LIN {X 0,Y 573.253,Z 273.707,A -85,B 0,C 180,E1 -2292.186,E2 -2292.186} C_VEL
LIN {X 0,Y 573.222,Z 273.707,A -85,B 0,C 180,E1 -2294.675,E2 -2294.675} C_VEL
LIN {X 0,Y 573.232,Z 273.706,A -85,B 0,C 180,E1 -2297.599,E2 -2297.599} C_VEL
LIN {X 0,Y 573.243,Z 273.707,A -85,B 0,C 180,E1 -2300.393,E2 -2300.393} C_VEL
LIN {X 0,Y 573.246,Z 273.706,A -85,B 0,C 180,E1 -2303.077,E2 -2303.077} C_VEL
LIN {X 0,Y 573.254,Z 273.702,A -85,B 0,C 180,E1 -2305.671,E2 -2305.671} C_VEL
LIN {X 0,Y 573.242,Z 273.706,A -85,B 0,C 180,E1 -2308.185,E2 -2308.185} C_VEL
LIN {X 0,Y 573.254,Z 273.705,A -85,B 0,C 180,E1 -2310.634,E2 -2310.634} C_VEL
LIN {X 0,Y 573.228,Z 273.706,A -85,B 0,C 180,E1 -2313.507,E2 -2313.507} C_VEL
LIN {X 0,Y 573.225,Z 273.705,A -85,B 0,C 180,E1 -2316.134,E2 -2316.134} C_VEL
LIN {X 0,Y 573.238,Z 273.704,A -85,B 0,C 180,E1 -2319.173,E2 -2319.173} C_VEL
LIN {X 0,Y 573.23,Z 273.707,A -85,B 0,C 180,E1 -2321.412,E2 -2321.412} C_VEL
LIN {X 0,Y 573.243,Z 273.704,A -85,B 0,C 180,E1 -2323.622,E2 -2323.622} C_VEL
LIN {X 0,Y 573.216,Z 273.708,A -85,B 0,C 180,E1 -2326.529,E2 -2326.529} C_VEL
LIN {X 0,Y 573.275,Z 273.699,A -85,B 0,C 180,E1 -2328.734,E2 -2328.734} C_VEL
LIN {X 0,Y 573.276,Z 273.698,A -85,B 0,C 180,E1 -2331.54,E2 -2331.54} C_VEL
LIN {X 0,Y 573.283,Z 273.698,A -85,B 0,C 180,E1 -2334.372,E2 -2334.372} C_VEL
LIN {X 0,Y 573.31,Z 273.694,A -85,B 0,C 180,E1 -2337.892,E2 -2337.892} C_VEL
LIN {X 0,Y 573.31,Z 273.695,A -85,B 0,C 180,E1 -2340.702,E2 -2340.702} C_VEL
LIN {X 0,Y 573.298,Z 273.699,A -85,B 0,C 180,E1 -2342.811,E2 -2342.811} C_VEL
LIN {X 0,Y 573.283,Z 273.699,A -85,B 0,C 180,E1 -2345.628,E2 -2345.628} C_VEL
LIN {X 0,Y 573.276,Z 273.698,A -85,B 0,C 180,E1 -2348.46,E2 -2348.46} C_VEL
LIN {X 0,Y 573.262,Z 273.7,A -85,B 0,C 180,E1 -2351.312,E2 -2351.312} C_VEL
LIN {X 0,Y 573.247,Z 273.703,A -85,B 0,C 180,E1 -2354.194,E2 -2354.194} C_VEL
LIN {X 0,Y 573.251,Z 273.704,A -85,B 0,C 180,E1 -2357.112,E2 -2357.112} C_VEL
LIN {X 0,Y 573.238,Z 273.707,A -85,B 0,C 180,E1 -2360.077,E2 -2360.077} C_VEL
LIN {X 0,Y 573.226,Z 273.705,A -85,B 0,C 180,E1 -2362.338,E2 -2362.338} C_VEL
LIN {X 0,Y 573.242,Z 273.704,A -85,B 0,C 180,E1 -2364.372,E2 -2364.372} C_VEL
LIN {X 0,Y 572.615,Z 273.786,A -85,B 0,C 180,E1 -2364.958,E2 -2364.958} C_VEL
LIN {X 0,Y 569.777,Z 274.144,A -85,B 0,C 180,E1 -2365.91,E2 -2365.91} C_VEL
LIN {X 0,Y 567.344,Z 274.445,A -85,B 0,C 180,E1 -2366.675,E2 -2366.675} C_VEL
LIN {X 0,Y 566.282,Z 274.573,A -85,B 0,C 180,E1 -2367.266,E2 -2367.266} C_VEL
LIN {X 0,Y 566.188,Z 274.583,A -85,B 0,C 180,E1 -2367.466,E2 -2367.466} C_VEL
LIN {X 0,Y 566.194,Z 274.58,A -85,B 0,C 180,E1 -2369.769,E2 -2369.769} C_VEL
LIN {X 0,Y 566.201,Z 274.582,A -85,B 0,C 180,E1 -2372.431,E2 -2372.431} C_VEL
LIN {X 0,Y 566.163,Z 274.588,A -85,B 0,C 180,E1 -2374.989,E2 -2374.989} C_VEL
LIN {X 0,Y 566.191,Z 274.581,A -85,B 0,C 180,E1 -2377.461,E2 -2377.461} C_VEL
LIN {X 0,Y 566.213,Z 274.58,A -85,B 0,C 180,E1 -2380.199,E2 -2380.199} C_VEL
LIN {X 0,Y 566.195,Z 274.584,A -85,B 0,C 180,E1 -2383.055,E2 -2383.055} C_VEL
LIN {X 0,Y 566.198,Z 274.586,A -85,B 0,C 180,E1 -2386.049,E2 -2386.049} C_VEL
LIN {X 0,Y 566.161,Z 274.589,A -85,B 0,C 180,E1 -2388.143,E2 -2388.143} C_VEL
LIN {X 0,Y 566.274,Z 277.89,A -85,B 0,C 180,E1 -2390.307,E2 -2390.307} C_VEL
LIN {X 0,Y 566.241,Z 283.039,A -85,B 0,C 180,E1 -2393.434,E2 -2393.434} C_VEL
LIN {X 0,Y 566.196,Z 287.886,A -85,B 0,C 180,E1 -2396.269,E2 -2396.269} C_VEL
LIN {X 0,Y 566.108,Z 292.591,A -85,B 0,C 180,E1 -2398.938,E2 -2398.938} C_VEL
LIN {X 0,Y 566.097,Z 297.844,A -85,B 0,C 180,E1 -2401.852,E2 -2401.852} C_VEL
LIN {X 0,Y 566.04,Z 303.736,A -85,B 0,C 180,E1 -2405.031,E2 -2405.031} C_VEL
LIN {X 0,Y 565.959,Z 308.198,A -85,B 0,C 180,E1 -2407.36,E2 -2407.36} C_VEL
LIN {X 0,Y 565.927,Z 314.163,A -85,B 0,C 180,E1 -2410.41,E2 -2410.41} C_VEL
LIN {X 0,Y 565.941,Z 317.901,A -85,B 0,C 180,E1 -2412.22,E2 -2412.22} C_VEL
LIN {X 0,Y 567.973,Z 327.367,A -85,B 0,C 180,E1 -2412.436,E2 -2412.436} C_VEL
LIN {X 0,Y 567.841,Z 342.313,A -85,B 0,C 180,E1 -2412.783,E2 -2412.783} C_VEL
LIN {X 0,Y 567.585,Z 357.472,A -85,B 0,C 180,E1 -2413.285,E2 -2413.285} C_VEL
LIN {X 0,Y 567.356,Z 371.746,A -85,B 0,C 180,E1 -2413.909,E2 -2413.909} C_VEL
LIN {X 0,Y 567.155,Z 385.053,A -85,B 0,C 180,E1 -2414.641,E2 -2414.641} C_VEL
LIN {X 0,Y 566.917,Z 397.983,A -85,B 0,C 180,E1 -2415.508,E2 -2415.508} C_VEL
LIN {X 0,Y 566.65,Z 410.894,A -85,B 0,C 180,E1 -2416.553,E2 -2416.553} C_VEL
LIN {X 0,Y 566.462,Z 422.089,A -85,B 0,C 180,E1 -2417.643,E2 -2417.643} C_VEL
LIN {X 0,Y 566.263,Z 432.181,A -85,B 0,C 180,E1 -2418.81,E2 -2418.81} C_VEL
LIN {X 0,Y 566.132,Z 442.007,A -85,B 0,C 180,E1 -2420.172,E2 -2420.172} C_VEL
LIN {X 0,Y 566.063,Z 449.498,A -85,B 0,C 180,E1 -2421.432,E2 -2421.432} C_VEL
LIN {X 0,Y 565.975,Z 456.501,A -85,B 0,C 180,E1 -2422.867,E2 -2422.867} C_VEL
LIN {X 0,Y 565.982,Z 462.009,A -85,B 0,C 180,E1 -2424.299,E2 -2424.299} C_VEL
LIN {X 0,Y 565.913,Z 466.178,A -85,B 0,C 180,E1 -2425.727,E2 -2425.727} C_VEL
LIN {X 0,Y 565.872,Z 469.114,A -85,B 0,C 180,E1 -2427.153,E2 -2427.153} C_VEL
LIN {X 0,Y 565.842,Z 470.88,A -85,B 0,C 180,E1 -2428.577,E2 -2428.577} C_VEL
LIN {X 0,Y 565.837,Z 471.496,A -85,B 0,C 180,E1 -2430,E2 -2430} C_VEL
LIN {X 0,Y 565.843,Z 470.941,A -85,B 0,C 180,E1 -2431.424,E2 -2431.424} C_VEL
LIN {X 0,Y 565.874,Z 469.258,A -85,B 0,C 180,E1 -2432.848,E2 -2432.848} C_VEL
LIN {X 0,Y 565.913,Z 466.402,A -85,B 0,C 180,E1 -2434.273,E2 -2434.273} C_VEL
LIN {X 0,Y 565.975,Z 462.317,A -85,B 0,C 180,E1 -2435.701,E2 -2435.701} C_VEL
LIN {X 0,Y 565.975,Z 456.903,A -85,B 0,C 180,E1 -2437.133,E2 -2437.133} C_VEL
LIN {X 0,Y 566.061,Z 450.002,A -85,B 0,C 180,E1 -2438.568,E2 -2438.568} C_VEL
LIN {X 0,Y 566.177,Z 441.394,A -85,B 0,C 180,E1 -2440.008,E2 -2440.008} C_VEL
LIN {X 0,Y 566.25,Z 432.951,A -85,B 0,C 180,E1 -2441.183,E2 -2441.183} C_VEL
LIN {X 0,Y 566.43,Z 422.914,A -85,B 0,C 180,E1 -2442.359,E2 -2442.359} C_VEL
LIN {X 0,Y 566.669,Z 410.869,A -85,B 0,C 180,E1 -2443.538,E2 -2443.538} C_VEL
LIN {X 0,Y 566.88,Z 399.267,A -85,B 0,C 180,E1 -2444.487,E2 -2444.487} C_VEL
LIN {X 0,Y 567.094,Z 386.474,A -85,B 0,C 180,E1 -2445.361,E2 -2445.361} C_VEL
LIN {X 0,Y 567.343,Z 373.462,A -85,B 0,C 180,E1 -2446.092,E2 -2446.092} C_VEL
LIN {X 0,Y 567.554,Z 359.278,A -85,B 0,C 180,E1 -2446.732,E2 -2446.732} C_VEL
LIN {X 0,Y 567.766,Z 344.75,A -85,B 0,C 180,E1 -2447.235,E2 -2447.235} C_VEL
LIN {X 0,Y 567.948,Z 329.926,A -85,B 0,C 180,E1 -2447.602,E2 -2447.602} C_VEL
LIN {X 0,Y 567.689,Z 325.292,A -85,B 0,C 180,E1 -2447.701,E2 -2447.701} C_VEL
LIN {X 0,Y 565.905,Z 317.734,A -85,B 0,C 180,E1 -2447.882,E2 -2447.882} C_VEL
LIN {X 0,Y 565.906,Z 312.848,A -85,B 0,C 180,E1 -2450.349,E2 -2450.349} C_VEL
LIN {X 0,Y 565.99,Z 306.879,A -85,B 0,C 180,E1 -2453.412,E2 -2453.412} C_VEL
LIN {X 0,Y 566.009,Z 302.424,A -85,B 0,C 180,E1 -2455.759,E2 -2455.759} C_VEL
LIN {X 0,Y 566.083,Z 297.941,A -85,B 0,C 180,E1 -2458.179,E2 -2458.179} C_VEL
LIN {X 0,Y 566.117,Z 292.097,A -85,B 0,C 180,E1 -2461.426,E2 -2461.426} C_VEL
LIN {X 0,Y 566.202,Z 287.652,A -85,B 0,C 180,E1 -2463.956,E2 -2463.956} C_VEL
LIN {X 0,Y 566.244,Z 283.188,A -85,B 0,C 180,E1 -2466.566,E2 -2466.566} C_VEL
LIN {X 0,Y 566.276,Z 278.037,A -85,B 0,C 180,E1 -2469.693,E2 -2469.693} C_VEL
LIN {X 0,Y 566.169,Z 274.608,A -85,B 0,C 180,E1 -2471.858,E2 -2471.858} C_VEL
LIN {X 0,Y 566.196,Z 274.586,A -85,B 0,C 180,E1 -2474.035,E2 -2474.035} C_VEL
LIN {X 0,Y 566.199,Z 274.585,A -85,B 0,C 180,E1 -2477.083,E2 -2477.083} C_VEL
LIN {X 0,Y 566.221,Z 274.584,A -85,B 0,C 180,E1 -2480.313,E2 -2480.313} C_VEL
LIN {X 0,Y 566.191,Z 274.587,A -85,B 0,C 180,E1 -2483.429,E2 -2483.429} C_VEL
LIN {X 0,Y 566.208,Z 274.584,A -85,B 0,C 180,E1 -2486.266,E2 -2486.266} C_VEL
LIN {X 0,Y 566.196,Z 274.582,A -85,B 0,C 180,E1 -2488.922,E2 -2488.922} C_VEL
LIN {X 0,Y 566.183,Z 274.582,A -85,B 0,C 180,E1 -2491.856,E2 -2491.856} C_VEL
LIN {X 0,Y 566.205,Z 274.583,A -85,B 0,C 180,E1 -2494.25,E2 -2494.25} C_VEL
LIN {X 0,Y 566.189,Z 274.583,A -85,B 0,C 180,E1 -2496.713,E2 -2496.713} C_VEL
LIN {X 0,Y 566.198,Z 274.581,A -85,B 0,C 180,E1 -2499.662,E2 -2499.662} C_VEL
LIN {X 0,Y 566.199,Z 274.581,A -85,B 0,C 180,E1 -2502.668,E2 -2502.668} C_VEL
LIN {X 0,Y 566.209,Z 274.579,A -85,B 0,C 180,E1 -2505.626,E2 -2505.626} C_VEL
LIN {X 0,Y 566.231,Z 274.576,A -85,B 0,C 180,E1 -2508.675,E2 -2508.675} C_VEL
LIN {X 0,Y 566.223,Z 274.577,A -85,B 0,C 180,E1 -2511.434,E2 -2511.434} C_VEL
LIN {X 0,Y 566.251,Z 274.576,A -85,B 0,C 180,E1 -2514.302,E2 -2514.302} C_VEL
LIN {X 0,Y 566.283,Z 274.57,A -85,B 0,C 180,E1 -2517.866,E2 -2517.866} C_VEL
LIN {X 0,Y 566.284,Z 274.57,A -85,B 0,C 180,E1 -2520.711,E2 -2520.711} C_VEL
LIN {X 0,Y 566.267,Z 274.575,A -85,B 0,C 180,E1 -2522.846,E2 -2522.846} C_VEL
LIN {X 0,Y 566.253,Z 274.574,A -85,B 0,C 180,E1 -2525.698,E2 -2525.698} C_VEL
LIN {X 0,Y 566.222,Z 274.578,A -85,B 0,C 180,E1 -2528.566,E2 -2528.566} C_VEL
LIN {X 0,Y 566.238,Z 274.576,A -85,B 0,C 180,E1 -2531.454,E2 -2531.454} C_VEL
LIN {X 0,Y 566.217,Z 274.578,A -85,B 0,C 180,E1 -2534.502,E2 -2534.502} C_VEL
LIN {X 0,Y 566.2,Z 274.581,A -85,B 0,C 180,E1 -2537.332,E2 -2537.332} C_VEL
LIN {X 0,Y 566.199,Z 274.582,A -85,B 0,C 180,E1 -2540.338,E2 -2540.338} C_VEL
LIN {X 0,Y 566.168,Z 274.586,A -85,B 0,C 180,E1 -2543.282,E2 -2543.282} C_VEL
LIN {X 0,Y 566.211,Z 274.581,A -85,B 0,C 180,E1 -2545.749,E2 -2545.749} C_VEL
LIN {X 0,Y 566.199,Z 274.581,A -85,B 0,C 180,E1 -2548.202,E2 -2548.202} C_VEL
LIN {X 0,Y 566.192,Z 274.583,A -85,B 0,C 180,E1 -2551.077,E2 -2551.077} C_VEL
LIN {X 0,Y 566.207,Z 274.586,A -85,B 0,C 180,E1 -2553.734,E2 -2553.734} C_VEL
LIN {X 0,Y 566.189,Z 274.587,A -85,B 0,C 180,E1 -2556.571,E2 -2556.571} C_VEL
LIN {X 0,Y 566.22,Z 274.583,A -85,B 0,C 180,E1 -2559.687,E2 -2559.687} C_VEL
LIN {X 0,Y 566.193,Z 274.587,A -85,B 0,C 180,E1 -2562.917,E2 -2562.917} C_VEL
LIN {X 0,Y 566.197,Z 274.588,A -85,B 0,C 180,E1 -2566.049,E2 -2566.049} C_VEL
LIN {X 0,Y 566.226,Z 274.656,A -85,B 0,C 180,E1 -2567.794,E2 -2567.794} C_VEL
LIN {X 0,Y 566.433,Z 278.416,A -85,B 0,C 180,E1 -2569.821,E2 -2569.821} C_VEL
LIN {X 0,Y 566.347,Z 283.788,A -85,B 0,C 180,E1 -2572.58,E2 -2572.58} C_VEL
LIN {X 0,Y 566.277,Z 289.058,A -85,B 0,C 180,E1 -2575.187,E2 -2575.187} C_VEL
LIN {X 0,Y 566.25,Z 294.398,A -85,B 0,C 180,E1 -2577.745,E2 -2577.745} C_VEL
LIN {X 0,Y 566.149,Z 301.557,A -85,B 0,C 180,E1 -2581.044,E2 -2581.044} C_VEL
LIN {X 0,Y 566.097,Z 306.924,A -85,B 0,C 180,E1 -2583.453,E2 -2583.453} C_VEL
LIN {X 0,Y 566.033,Z 312.275,A -85,B 0,C 180,E1 -2585.812,E2 -2585.812} C_VEL
LIN {X 0,Y 566.019,Z 319.366,A -85,B 0,C 180,E1 -2588.895,E2 -2588.895} C_VEL
LIN {X 0,Y 565.972,Z 326.457,A -85,B 0,C 180,E1 -2591.914,E2 -2591.914} C_VEL
LIN {X 0,Y 565.98,Z 327.042,A -85,B 0,C 180,E1 -2592.161,E2 -2592.161} C_VEL
LIN {X 0,Y 567.973,Z 335.917,A -85,B 0,C 180,E1 -2592.363,E2 -2592.363} C_VEL
LIN {X 0,Y 567.838,Z 351.705,A -85,B 0,C 180,E1 -2592.72,E2 -2592.72} C_VEL
LIN {X 0,Y 567.604,Z 367.239,A -85,B 0,C 180,E1 -2593.231,E2 -2593.231} C_VEL
LIN {X 0,Y 567.384,Z 380.771,A -85,B 0,C 180,E1 -2593.817,E2 -2593.817} C_VEL
LIN {X 0,Y 567.15,Z 394.244,A -85,B 0,C 180,E1 -2594.548,E2 -2594.548} C_VEL
LIN {X 0,Y 566.927,Z 406.797,A -85,B 0,C 180,E1 -2595.379,E2 -2595.379} C_VEL
LIN {X 0,Y 566.672,Z 419.29,A -85,B 0,C 180,E1 -2596.37,E2 -2596.37} C_VEL
LIN {X 0,Y 566.491,Z 430.748,A -85,B 0,C 180,E1 -2597.461,E2 -2597.461} C_VEL
LIN {X 0,Y 566.268,Z 441.312,A -85,B 0,C 180,E1 -2598.659,E2 -2598.659} C_VEL
LIN {X 0,Y 566.208,Z 449.856,A -85,B 0,C 180,E1 -2599.812,E2 -2599.812} C_VEL
LIN {X 0,Y 566.057,Z 457.733,A -85,B 0,C 180,E1 -2601.072,E2 -2601.072} C_VEL
LIN {X 0,Y 565.997,Z 465.089,A -85,B 0,C 180,E1 -2602.508,E2 -2602.508} C_VEL
LIN {X 0,Y 565.959,Z 470.922,A -85,B 0,C 180,E1 -2603.941,E2 -2603.941} C_VEL
LIN {X 0,Y 565.867,Z 474.385,A -85,B 0,C 180,E1 -2605.012,E2 -2605.012} C_VEL
LIN {X 0,Y 565.91,Z 477.889,A -85,B 0,C 180,E1 -2606.44,E2 -2606.44} C_VEL
LIN {X 0,Y 565.839,Z 480.192,A -85,B 0,C 180,E1 -2607.864,E2 -2607.864} C_VEL
LIN {X 0,Y 565.837,Z 481.349,A -85,B 0,C 180,E1 -2609.288,E2 -2609.288} C_VEL
LIN {X 0,Y 565.837,Z 481.349,A -85,B 0,C 180,E1 -2610.711,E2 -2610.711} C_VEL
LIN {X 0,Y 565.839,Z 480.191,A -85,B 0,C 180,E1 -2612.135,E2 -2612.135} C_VEL
LIN {X 0,Y 565.91,Z 477.888,A -85,B 0,C 180,E1 -2613.56,E2 -2613.56} C_VEL
LIN {X 0,Y 565.866,Z 474.386,A -85,B 0,C 180,E1 -2614.987,E2 -2614.987} C_VEL
LIN {X 0,Y 565.942,Z 469.61,A -85,B 0,C 180,E1 -2616.417,E2 -2616.417} C_VEL
LIN {X 0,Y 566.014,Z 463.425,A -85,B 0,C 180,E1 -2617.85,E2 -2617.85} C_VEL
LIN {X 0,Y 566.071,Z 455.65,A -85,B 0,C 180,E1 -2619.288,E2 -2619.288} C_VEL
LIN {X 0,Y 566.239,Z 447.372,A -85,B 0,C 180,E1 -2620.548,E2 -2620.548} C_VEL
LIN {X 0,Y 566.366,Z 437.395,A -85,B 0,C 180,E1 -2621.814,E2 -2621.814} C_VEL
LIN {X 0,Y 566.585,Z 427.193,A -85,B 0,C 180,E1 -2622.901,E2 -2622.901} C_VEL
LIN {X 0,Y 566.799,Z 415.025,A -85,B 0,C 180,E1 -2623.992,E2 -2623.992} C_VEL
LIN {X 0,Y 567.038,Z 402.348,A -85,B 0,C 180,E1 -2624.936,E2 -2624.936} C_VEL
LIN {X 0,Y 567.215,Z 389.523,A -85,B 0,C 180,E1 -2625.726,E2 -2625.726} C_VEL
LIN {X 0,Y 567.468,Z 374.842,A -85,B 0,C 180,E1 -2626.457,E2 -2626.457} C_VEL
LIN {X 0,Y 567.761,Z 359.722,A -85,B 0,C 180,E1 -2627.036,E2 -2627.036} C_VEL
LIN {X 0,Y 567.89,Z 344.457,A -85,B 0,C 180,E1 -2627.464,E2 -2627.464} C_VEL
LIN {X 0,Y 567.77,Z 334.752,A -85,B 0,C 180,E1 -2627.662,E2 -2627.662} C_VEL
LIN {X 0,Y 565.973,Z 327.038,A -85,B 0,C 180,E1 -2627.841,E2 -2627.841} C_VEL
LIN {X 0,Y 565.979,Z 321.14,A -85,B 0,C 180,E1 -2630.345,E2 -2630.345} C_VEL
LIN {X 0,Y 566.043,Z 314.412,A -85,B 0,C 180,E1 -2633.251,E2 -2633.251} C_VEL
LIN {X 0,Y 566.056,Z 308.708,A -85,B 0,C 180,E1 -2635.756,E2 -2635.756} C_VEL
LIN {X 0,Y 566.131,Z 303.233,A -85,B 0,C 180,E1 -2638.188,E2 -2638.188} C_VEL
LIN {X 0,Y 566.187,Z 296.931,A -85,B 0,C 180,E1 -2641.076,E2 -2641.076} C_VEL
LIN {X 0,Y 566.277,Z 290.828,A -85,B 0,C 180,E1 -2643.95,E2 -2643.95} C_VEL
LIN {X 0,Y 566.327,Z 285.511,A -85,B 0,C 180,E1 -2646.559,E2 -2646.559} C_VEL
LIN {X 0,Y 566.389,Z 280.186,A -85,B 0,C 180,E1 -2649.258,E2 -2649.258} C_VEL
LIN {X 0,Y 566.41,Z 276.644,A -85,B 0,C 180,E1 -2651.118,E2 -2651.118} C_VEL
LIN {X 0,Y 566.198,Z 274.586,A -85,B 0,C 180,E1 -2652.328,E2 -2652.328} C_VEL
LIN {X 0,Y 566.168,Z 274.586,A -85,B 0,C 180,E1 -2655.035,E2 -2655.035} C_VEL
LIN {X 0,Y 566.181,Z 274.583,A -85,B 0,C 180,E1 -2657.91,E2 -2657.91} C_VEL
LIN {X 0,Y 566.218,Z 274.579,A -85,B 0,C 180,E1 -2660.727,E2 -2660.727} C_VEL
LIN {X 0,Y 566.186,Z 274.587,A -85,B 0,C 180,E1 -2663.429,E2 -2663.429} C_VEL
LIN {X 0,Y 566.203,Z 274.586,A -85,B 0,C 180,E1 -2666.266,E2 -2666.266} C_VEL
LIN {X 0,Y 566.192,Z 274.583,A -85,B 0,C 180,E1 -2668.922,E2 -2668.922} C_VEL
LIN {X 0,Y 566.182,Z 274.583,A -85,B 0,C 180,E1 -2671.856,E2 -2671.856} C_VEL
LIN {X 0,Y 566.208,Z 274.582,A -85,B 0,C 180,E1 -2674.251,E2 -2674.251} C_VEL
LIN {X 0,Y 566.184,Z 274.584,A -85,B 0,C 180,E1 -2676.713,E2 -2676.713} C_VEL
LIN {X 0,Y 566.2,Z 274.581,A -85,B 0,C 180,E1 -2679.662,E2 -2679.662} C_VEL
LIN {X 0,Y 566.201,Z 274.582,A -85,B 0,C 180,E1 -2681.922,E2 -2681.922} C_VEL
LIN {X 0,Y 566.192,Z 274.582,A -85,B 0,C 180,E1 -2684.152,E2 -2684.152} C_VEL
LIN {X 0,Y 566.178,Z 274.587,A -85,B 0,C 180,E1 -2686.358,E2 -2686.358} C_VEL
LIN {X 0,Y 566.267,Z 274.572,A -85,B 0,C 180,E1 -2688.654,E2 -2688.654} C_VEL
LIN {X 0,Y 566.22,Z 274.578,A -85,B 0,C 180,E1 -2691.434,E2 -2691.434} C_VEL
LIN {X 0,Y 566.25,Z 274.575,A -85,B 0,C 180,E1 -2694.302,E2 -2694.302} C_VEL
LIN {X 0,Y 566.28,Z 274.57,A -85,B 0,C 180,E1 -2697.866,E2 -2697.866} C_VEL
LIN {X 0,Y 566.282,Z 274.57,A -85,B 0,C 180,E1 -2700.711,E2 -2700.711} C_VEL
LIN {X 0,Y 566.265,Z 274.575,A -85,B 0,C 180,E1 -2702.846,E2 -2702.846} C_VEL
LIN {X 0,Y 566.25,Z 274.575,A -85,B 0,C 180,E1 -2705.698,E2 -2705.698} C_VEL
LIN {X 0,Y 566.22,Z 274.577,A -85,B 0,C 180,E1 -2708.566,E2 -2708.566} C_VEL
LIN {X 0,Y 566.233,Z 274.575,A -85,B 0,C 180,E1 -2711.455,E2 -2711.455} C_VEL
LIN {X 0,Y 566.212,Z 274.578,A -85,B 0,C 180,E1 -2714.502,E2 -2714.502} C_VEL
LIN {X 0,Y 566.196,Z 274.581,A -85,B 0,C 180,E1 -2717.332,E2 -2717.332} C_VEL
LIN {X 0,Y 566.201,Z 274.582,A -85,B 0,C 180,E1 -2719.581,E2 -2719.581} C_VEL
LIN {X 0,Y 566.184,Z 274.583,A -85,B 0,C 180,E1 -2721.863,E2 -2721.863} C_VEL
LIN {X 0,Y 566.228,Z 274.577,A -85,B 0,C 180,E1 -2724.961,E2 -2724.961} C_VEL
LIN {X 0,Y 566.188,Z 274.583,A -85,B 0,C 180,E1 -2727.466,E2 -2727.466} C_VEL
LIN {X 0,Y 565.5,Z 274.668,A -85,B 0,C 180,E1 -2728.06,E2 -2728.06} C_VEL
LIN {X 0,Y 562.638,Z 275.029,A -85,B 0,C 180,E1 -2729.024,E2 -2729.024} C_VEL
LIN {X 0,Y 560.239,Z 275.325,A -85,B 0,C 180,E1 -2729.8,E2 -2729.8} C_VEL
LIN {X 0,Y 559.217,Z 275.453,A -85,B 0,C 180,E1 -2730.398,E2 -2730.398} C_VEL
LIN {X 0,Y 559.138,Z 275.459,A -85,B 0,C 180,E1 -2730.601,E2 -2730.601} C_VEL
LIN {X 0,Y 559.167,Z 275.456,A -85,B 0,C 180,E1 -2732.715,E2 -2732.715} C_VEL
LIN {X 0,Y 559.111,Z 275.467,A -85,B 0,C 180,E1 -2735.325,E2 -2735.325} C_VEL
LIN {X 0,Y 559.131,Z 275.464,A -85,B 0,C 180,E1 -2738.018,E2 -2738.018} C_VEL
LIN {X 0,Y 559.167,Z 275.457,A -85,B 0,C 180,E1 -2740.812,E2 -2740.812} C_VEL
LIN {X 0,Y 559.136,Z 275.46,A -85,B 0,C 180,E1 -2743.735,E2 -2743.735} C_VEL
LIN {X 0,Y 559.164,Z 275.459,A -85,B 0,C 180,E1 -2746.802,E2 -2746.802} C_VEL
LIN {X 0,Y 559.147,Z 275.623,A -85,B 0,C 180,E1 -2748.229,E2 -2748.229} C_VEL
LIN {X 0,Y 559.233,Z 278.609,A -85,B 0,C 180,E1 -2750.14,E2 -2750.14} C_VEL
LIN {X 0,Y 559.205,Z 283.072,A -85,B 0,C 180,E1 -2752.898,E2 -2752.898} C_VEL
LIN {X 0,Y 559.156,Z 288.374,A -85,B 0,C 180,E1 -2756.053,E2 -2756.053} C_VEL
LIN {X 0,Y 559.058,Z 293.453,A -85,B 0,C 180,E1 -2758.976,E2 -2758.976} C_VEL
LIN {X 0,Y 559.033,Z 298.218,A -85,B 0,C 180,E1 -2761.645,E2 -2761.645} C_VEL
LIN {X 0,Y 558.968,Z 304.094,A -85,B 0,C 180,E1 -2764.86,E2 -2764.86} C_VEL
LIN {X 0,Y 558.906,Z 308.201,A -85,B 0,C 180,E1 -2767.058,E2 -2767.058} C_VEL
LIN {X 0,Y 558.819,Z 312.673,A -85,B 0,C 180,E1 -2769.382,E2 -2769.382} C_VEL
LIN {X 0,Y 558.835,Z 317.783,A -85,B 0,C 180,E1 -2771.984,E2 -2771.984} C_VEL
LIN {X 0,Y 561.211,Z 327.633,A -85,B 0,C 180,E1 -2772.223,E2 -2772.223} C_VEL
LIN {X 0,Y 561.06,Z 342.105,A -85,B 0,C 180,E1 -2772.561,E2 -2772.561} C_VEL
LIN {X 0,Y 560.797,Z 356.783,A -85,B 0,C 180,E1 -2773.047,E2 -2773.047} C_VEL
LIN {X 0,Y 560.503,Z 371.755,A -85,B 0,C 180,E1 -2773.707,E2 -2773.707} C_VEL
LIN {X 0,Y 560.256,Z 385.065,A -85,B 0,C 180,E1 -2774.447,E2 -2774.447} C_VEL
LIN {X 0,Y 559.983,Z 398.395,A -85,B 0,C 180,E1 -2775.354,E2 -2775.354} C_VEL
LIN {X 0,Y 559.691,Z 410.901,A -85,B 0,C 180,E1 -2776.383,E2 -2776.383} C_VEL
LIN {X 0,Y 559.486,Z 422.095,A -85,B 0,C 180,E1 -2777.486,E2 -2777.486} C_VEL
LIN {X 0,Y 559.228,Z 432.79,A -85,B 0,C 180,E1 -2778.743,E2 -2778.743} C_VEL
LIN {X 0,Y 559.095,Z 442.01,A -85,B 0,C 180,E1 -2780.047,E2 -2780.047} C_VEL
LIN {X 0,Y 559.002,Z 449.5,A -85,B 0,C 180,E1 -2781.323,E2 -2781.323} C_VEL
LIN {X 0,Y 558.9,Z 456.503,A -85,B 0,C 180,E1 -2782.777,E2 -2782.777} C_VEL
LIN {X 0,Y 558.888,Z 462.012,A -85,B 0,C 180,E1 -2784.227,E2 -2784.227} C_VEL
LIN {X 0,Y 558.808,Z 466.18,A -85,B 0,C 180,E1 -2785.673,E2 -2785.673} C_VEL
LIN {X 0,Y 558.793,Z 469.114,A -85,B 0,C 180,E1 -2787.117,E2 -2787.117} C_VEL
LIN {X 0,Y 558.742,Z 470.88,A -85,B 0,C 180,E1 -2788.559,E2 -2788.559} C_VEL
LIN {X 0,Y 558.738,Z 471.496,A -85,B 0,C 180,E1 -2790,E2 -2790} C_VEL
LIN {X 0,Y 558.743,Z 470.94,A -85,B 0,C 180,E1 -2791.442,E2 -2791.442} C_VEL
LIN {X 0,Y 558.795,Z 469.256,A -85,B 0,C 180,E1 -2792.884,E2 -2792.884} C_VEL
LIN {X 0,Y 558.808,Z 466.402,A -85,B 0,C 180,E1 -2794.328,E2 -2794.328} C_VEL
LIN {X 0,Y 558.881,Z 462.315,A -85,B 0,C 180,E1 -2795.774,E2 -2795.774} C_VEL
LIN {X 0,Y 558.901,Z 456.9,A -85,B 0,C 180,E1 -2797.224,E2 -2797.224} C_VEL
LIN {X 0,Y 559.001,Z 449.999,A -85,B 0,C 180,E1 -2798.677,E2 -2798.677} C_VEL
LIN {X 0,Y 559.092,Z 442.57,A -85,B 0,C 180,E1 -2799.953,E2 -2799.953} C_VEL
LIN {X 0,Y 559.215,Z 433.509,A -85,B 0,C 180,E1 -2801.25,E2 -2801.25} C_VEL
LIN {X 0,Y 559.44,Z 422.908,A -85,B 0,C 180,E1 -2802.516,E2 -2802.516} C_VEL
LIN {X 0,Y 559.696,Z 410.863,A -85,B 0,C 180,E1 -2803.71,E2 -2803.71} C_VEL
LIN {X 0,Y 559.974,Z 398.309,A -85,B 0,C 180,E1 -2804.742,E2 -2804.742} C_VEL
LIN {X 0,Y 560.266,Z 385.002,A -85,B 0,C 180,E1 -2805.646,E2 -2805.646} C_VEL
LIN {X 0,Y 560.532,Z 371.682,A -85,B 0,C 180,E1 -2806.386,E2 -2806.386} C_VEL
LIN {X 0,Y 560.823,Z 357.425,A -85,B 0,C 180,E1 -2807.015,E2 -2807.015} C_VEL
LIN {X 0,Y 561.063,Z 342.029,A -85,B 0,C 180,E1 -2807.531,E2 -2807.531} C_VEL
LIN {X 0,Y 561.032,Z 326.98,A -85,B 0,C 180,E1 -2807.887,E2 -2807.887} C_VEL
LIN {X 0,Y 558.86,Z 317.738,A -85,B 0,C 180,E1 -2808.113,E2 -2808.113} C_VEL
LIN {X 0,Y 558.823,Z 312.846,A -85,B 0,C 180,E1 -2810.618,E2 -2810.618} C_VEL
LIN {X 0,Y 558.914,Z 306.891,A -85,B 0,C 180,E1 -2813.727,E2 -2813.727} C_VEL
LIN {X 0,Y 558.931,Z 302.458,A -85,B 0,C 180,E1 -2816.109,E2 -2816.109} C_VEL
LIN {X 0,Y 559.026,Z 298.029,A -85,B 0,C 180,E1 -2818.537,E2 -2818.537} C_VEL
LIN {X 0,Y 559.075,Z 293.196,A -85,B 0,C 180,E1 -2821.261,E2 -2821.261} C_VEL
LIN {X 0,Y 559.158,Z 288.526,A -85,B 0,C 180,E1 -2823.948,E2 -2823.948} C_VEL
LIN {X 0,Y 559.208,Z 283.221,A -85,B 0,C 180,E1 -2827.103,E2 -2827.103} C_VEL
LIN {X 0,Y 559.232,Z 278.604,A -85,B 0,C 180,E1 -2829.95,E2 -2829.95} C_VEL
LIN {X 0,Y 559.154,Z 275.761,A -85,B 0,C 180,E1 -2831.771,E2 -2831.771} C_VEL
LIN {X 0,Y 559.153,Z 275.464,A -85,B 0,C 180,E1 -2832.744,E2 -2832.744} C_VEL
LIN {X 0,Y 559.152,Z 275.465,A -85,B 0,C 180,E1 -2835.76,E2 -2835.76} C_VEL
LIN {X 0,Y 559.158,Z 275.458,A -85,B 0,C 180,E1 -2838.229,E2 -2838.229} C_VEL
LIN {X 0,Y 559.177,Z 275.455,A -85,B 0,C 180,E1 -2841.191,E2 -2841.191} C_VEL
LIN {X 0,Y 559.121,Z 275.464,A -85,B 0,C 180,E1 -2843.788,E2 -2843.788} C_VEL
LIN {X 0,Y 559.16,Z 275.463,A -85,B 0,C 180,E1 -2846.425,E2 -2846.425} C_VEL
LIN {X 0,Y 559.16,Z 275.458,A -85,B 0,C 180,E1 -2848.981,E2 -2848.981} C_VEL
LIN {X 0,Y 559.13,Z 275.461,A -85,B 0,C 180,E1 -2851.625,E2 -2851.625} C_VEL
LIN {X 0,Y 559.169,Z 275.46,A -85,B 0,C 180,E1 -2853.902,E2 -2853.902} C_VEL
LIN {X 0,Y 559.154,Z 275.458,A -85,B 0,C 180,E1 -2856.567,E2 -2856.567} C_VEL
LIN {X 0,Y 559.169,Z 275.456,A -85,B 0,C 180,E1 -2859.395,E2 -2859.395} C_VEL
LIN {X 0,Y 559.146,Z 275.464,A -85,B 0,C 180,E1 -2861.686,E2 -2861.686} C_VEL
LIN {X 0,Y 559.16,Z 275.456,A -85,B 0,C 180,E1 -2863.948,E2 -2863.948} C_VEL
LIN {X 0,Y 559.149,Z 275.463,A -85,B 0,C 180,E1 -2866.183,E2 -2866.183} C_VEL
LIN {X 0,Y 559.193,Z 275.456,A -85,B 0,C 180,E1 -2869.133,E2 -2869.133} C_VEL
LIN {X 0,Y 559.195,Z 275.454,A -85,B 0,C 180,E1 -2872.053,E2 -2872.053} C_VEL
LIN {X 0,Y 559.25,Z 275.447,A -85,B 0,C 180,E1 -2874.953,E2 -2874.953} C_VEL
LIN {X 0,Y 559.253,Z 275.445,A -85,B 0,C 180,E1 -2877.839,E2 -2877.839} C_VEL
LIN {X 0,Y 559.256,Z 275.445,A -85,B 0,C 180,E1 -2880.72,E2 -2880.72} C_VEL
LIN {X 0,Y 559.234,Z 275.451,A -85,B 0,C 180,E1 -2882.881,E2 -2882.881} C_VEL
LIN {X 0,Y 559.22,Z 275.451,A -85,B 0,C 180,E1 -2885.77,E2 -2885.77} C_VEL
LIN {X 0,Y 559.182,Z 275.455,A -85,B 0,C 180,E1 -2888.674,E2 -2888.674} C_VEL
LIN {X 0,Y 559.201,Z 275.452,A -85,B 0,C 180,E1 -2891.6,E2 -2891.6} C_VEL
LIN {X 0,Y 559.176,Z 275.455,A -85,B 0,C 180,E1 -2894.588,E2 -2894.588} C_VEL
LIN {X 0,Y 559.159,Z 275.457,A -85,B 0,C 180,E1 -2897.557,E2 -2897.557} C_VEL
LIN {X 0,Y 559.159,Z 275.462,A -85,B 0,C 180,E1 -2899.838,E2 -2899.838} C_VEL
LIN {X 0,Y 559.134,Z 275.46,A -85,B 0,C 180,E1 -2902.153,E2 -2902.153} C_VEL
LIN {X 0,Y 559.172,Z 275.456,A -85,B 0,C 180,E1 -2905.298,E2 -2905.298} C_VEL
LIN {X 0,Y 559.133,Z 275.465,A -85,B 0,C 180,E1 -2907.715,E2 -2907.715} C_VEL
LIN {X 0,Y 559.145,Z 275.461,A -85,B 0,C 180,E1 -2910.183,E2 -2910.183} C_VEL
LIN {X 0,Y 559.155,Z 275.46,A -85,B 0,C 180,E1 -2912.715,E2 -2912.715} C_VEL
LIN {X 0,Y 559.114,Z 275.469,A -85,B 0,C 180,E1 -2915.325,E2 -2915.325} C_VEL
LIN {X 0,Y 559.133,Z 275.465,A -85,B 0,C 180,E1 -2918.017,E2 -2918.017} C_VEL
LIN {X 0,Y 559.151,Z 275.46,A -85,B 0,C 180,E1 -2920.813,E2 -2920.813} C_VEL
LIN {X 0,Y 559.138,Z 275.462,A -85,B 0,C 180,E1 -2923.734,E2 -2923.734} C_VEL
LIN {X 0,Y 559.144,Z 275.463,A -85,B 0,C 180,E1 -2926.804,E2 -2926.804} C_VEL
LIN {X 0,Y 559.184,Z 275.6,A -85,B 0,C 180,E1 -2927.669,E2 -2927.669} C_VEL
LIN {X 0,Y 559.427,Z 278.384,A -85,B 0,C 180,E1 -2929.212,E2 -2929.212} C_VEL
LIN {X 0,Y 559.356,Z 283.704,A -85,B 0,C 180,E1 -2932.001,E2 -2932.001} C_VEL
LIN {X 0,Y 559.267,Z 289.196,A -85,B 0,C 180,E1 -2934.768,E2 -2934.768} C_VEL
LIN {X 0,Y 559.214,Z 294.5,A -85,B 0,C 180,E1 -2937.355,E2 -2937.355} C_VEL
LIN {X 0,Y 559.097,Z 300.458,A -85,B 0,C 180,E1 -2940.152,E2 -2940.152} C_VEL
LIN {X 0,Y 559.075,Z 305.101,A -85,B 0,C 180,E1 -2942.282,E2 -2942.282} C_VEL
LIN {X 0,Y 558.973,Z 312.252,A -85,B 0,C 180,E1 -2945.486,E2 -2945.486} C_VEL
LIN {X 0,Y 558.969,Z 319.366,A -85,B 0,C 180,E1 -2948.616,E2 -2948.616} C_VEL
LIN {X 0,Y 558.889,Z 326.457,A -85,B 0,C 180,E1 -2951.677,E2 -2951.677} C_VEL
LIN {X 0,Y 558.9,Z 327.138,A -85,B 0,C 180,E1 -2951.932,E2 -2951.932} C_VEL
LIN {X 0,Y 561.19,Z 337.488,A -85,B 0,C 180,E1 -2952.174,E2 -2952.174} C_VEL
LIN {X 0,Y 561.006,Z 352.811,A -85,B 0,C 180,E1 -2952.537,E2 -2952.537} C_VEL
LIN {X 0,Y 560.797,Z 367.547,A -85,B 0,C 180,E1 -2953.034,E2 -2953.034} C_VEL
LIN {X 0,Y 560.552,Z 380.774,A -85,B 0,C 180,E1 -2953.615,E2 -2953.615} C_VEL
LIN {X 0,Y 560.274,Z 394.247,A -85,B 0,C 180,E1 -2954.354,E2 -2954.354} C_VEL
LIN {X 0,Y 560.005,Z 407.508,A -85,B 0,C 180,E1 -2955.245,E2 -2955.245} C_VEL
LIN {X 0,Y 559.697,Z 420.35,A -85,B 0,C 180,E1 -2956.29,E2 -2956.29} C_VEL
LIN {X 0,Y 559.474,Z 432.508,A -85,B 0,C 180,E1 -2957.485,E2 -2957.485} C_VEL
LIN {X 0,Y 559.197,Z 443.241,A -85,B 0,C 180,E1 -2958.758,E2 -2958.758} C_VEL
LIN {X 0,Y 559.091,Z 452.294,A -85,B 0,C 180,E1 -2960.047,E2 -2960.047} C_VEL
LIN {X 0,Y 559.001,Z 459.75,A -85,B 0,C 180,E1 -2961.323,E2 -2961.323} C_VEL
LIN {X 0,Y 558.9,Z 466.701,A -85,B 0,C 180,E1 -2962.776,E2 -2962.776} C_VEL
LIN {X 0,Y 558.888,Z 472.161,A -85,B 0,C 180,E1 -2964.226,E2 -2964.226} C_VEL
LIN {X 0,Y 558.809,Z 476.291,A -85,B 0,C 180,E1 -2965.672,E2 -2965.672} C_VEL
LIN {X 0,Y 558.793,Z 479.186,A -85,B 0,C 180,E1 -2967.116,E2 -2967.116} C_VEL
LIN {X 0,Y 558.742,Z 480.911,A -85,B 0,C 180,E1 -2968.558,E2 -2968.558} C_VEL
LIN {X 0,Y 558.737,Z 481.5,A -85,B 0,C 180,E1 -2970,E2 -2970} C_VEL
LIN {X 0,Y 558.742,Z 480.91,A -85,B 0,C 180,E1 -2971.441,E2 -2971.441} C_VEL
LIN {X 0,Y 558.793,Z 479.184,A -85,B 0,C 180,E1 -2972.883,E2 -2972.883} C_VEL
LIN {X 0,Y 558.808,Z 476.29,A -85,B 0,C 180,E1 -2974.327,E2 -2974.327} C_VEL
LIN {X 0,Y 558.888,Z 472.165,A -85,B 0,C 180,E1 -2975.773,E2 -2975.773} C_VEL
LIN {X 0,Y 558.899,Z 466.703,A -85,B 0,C 180,E1 -2977.224,E2 -2977.224} C_VEL
LIN {X 0,Y 559,Z 459.749,A -85,B 0,C 180,E1 -2978.677,E2 -2978.677} C_VEL
LIN {X 0,Y 559.091,Z 452.295,A -85,B 0,C 180,E1 -2979.953,E2 -2979.953} C_VEL
LIN {X 0,Y 559.227,Z 443.125,A -85,B 0,C 180,E1 -2981.257,E2 -2981.257} C_VEL
LIN {X 0,Y 559.474,Z 432.512,A -85,B 0,C 180,E1 -2982.514,E2 -2982.514} C_VEL
LIN {X 0,Y 559.7,Z 420.36,A -85,B 0,C 180,E1 -2983.71,E2 -2983.71} C_VEL
LIN {X 0,Y 560.002,Z 407.532,A -85,B 0,C 180,E1 -2984.753,E2 -2984.753} C_VEL
LIN {X 0,Y 560.273,Z 394.255,A -85,B 0,C 180,E1 -2985.645,E2 -2985.645} C_VEL
LIN {X 0,Y 560.539,Z 380.78,A -85,B 0,C 180,E1 -2986.385,E2 -2986.385} C_VEL
LIN {X 0,Y 560.839,Z 366.51,A -85,B 0,C 180,E1 -2987.007,E2 -2987.007} C_VEL
LIN {X 0,Y 561.052,Z 350.87,A -85,B 0,C 180,E1 -2987.519,E2 -2987.519} C_VEL
LIN {X 0,Y 561.042,Z 336.077,A -85,B 0,C 180,E1 -2987.859,E2 -2987.859} C_VEL
LIN {X 0,Y 558.919,Z 327.02,A -85,B 0,C 180,E1 -2988.081,E2 -2988.081} C_VEL
LIN {X 0,Y 558.967,Z 319.368,A -85,B 0,C 180,E1 -2991.384,E2 -2991.384} C_VEL
LIN {X 0,Y 558.971,Z 312.246,A -85,B 0,C 180,E1 -2994.513,E2 -2994.513} C_VEL
LIN {X 0,Y 559.034,Z 306.869,A -85,B 0,C 180,E1 -2996.909,E2 -2996.909} C_VEL
LIN {X 0,Y 559.085,Z 301.505,A -85,B 0,C 180,E1 -2999.356,E2 -2999.356} C_VEL
LIN {X 0,Y 559.174,Z 296.152,A -85,B 0,C 180,E1 -3001.861,E2 -3001.861} C_VEL
LIN {X 0,Y 559.242,Z 290.814,A -85,B 0,C 180,E1 -3004.437,E2 -3004.437} C_VEL
LIN {X 0,Y 559.326,Z 285.479,A -85,B 0,C 180,E1 -3007.093,E2 -3007.093} C_VEL
LIN {X 0,Y 559.394,Z 279.926,A -85,B 0,C 180,E1 -3009.97,E2 -3009.97} C_VEL
LIN {X 0,Y 559.332,Z 276.619,A -85,B 0,C 180,E1 -3011.754,E2 -3011.754} C_VEL
LIN {X 0,Y 559.178,Z 275.46,A -85,B 0,C 180,E1 -3012.412,E2 -3012.412} C_VEL
LIN {X 0,Y 559.134,Z 275.464,A -85,B 0,C 180,E1 -3015.26,E2 -3015.26} C_VEL
LIN {X 0,Y 559.157,Z 275.46,A -85,B 0,C 180,E1 -3018.229,E2 -3018.229} C_VEL
LIN {X 0,Y 559.173,Z 275.456,A -85,B 0,C 180,E1 -3021.19,E2 -3021.19} C_VEL
LIN {X 0,Y 559.116,Z 275.464,A -85,B 0,C 180,E1 -3023.788,E2 -3023.788} C_VEL
LIN {X 0,Y 559.155,Z 275.464,A -85,B 0,C 180,E1 -3026.425,E2 -3026.425} C_VEL
LIN {X 0,Y 559.156,Z 275.46,A -85,B 0,C 180,E1 -3028.981,E2 -3028.981} C_VEL
LIN {X 0,Y 559.136,Z 275.461,A -85,B 0,C 180,E1 -3031.623,E2 -3031.623} C_VEL
LIN {X 0,Y 559.173,Z 275.461,A -85,B 0,C 180,E1 -3033.903,E2 -3033.903} C_VEL
LIN {X 0,Y 559.149,Z 275.459,A -85,B 0,C 180,E1 -3036.567,E2 -3036.567} C_VEL
LIN {X 0,Y 559.168,Z 275.456,A -85,B 0,C 180,E1 -3039.395,E2 -3039.395} C_VEL
LIN {X 0,Y 559.147,Z 275.464,A -85,B 0,C 180,E1 -3041.686,E2 -3041.686} C_VEL
LIN {X 0,Y 559.156,Z 275.458,A -85,B 0,C 180,E1 -3043.948,E2 -3043.948} C_VEL
LIN {X 0,Y 559.152,Z 275.463,A -85,B 0,C 180,E1 -3046.184,E2 -3046.184} C_VEL
LIN {X 0,Y 559.204,Z 275.455,A -85,B 0,C 180,E1 -3049.134,E2 -3049.134} C_VEL
LIN {X 0,Y 559.19,Z 275.455,A -85,B 0,C 180,E1 -3052.053,E2 -3052.053} C_VEL
LIN {X 0,Y 559.249,Z 275.446,A -85,B 0,C 180,E1 -3054.953,E2 -3054.953} C_VEL
LIN {X 0,Y 559.251,Z 275.445,A -85,B 0,C 180,E1 -3057.839,E2 -3057.839} C_VEL
LIN {X 0,Y 559.253,Z 275.445,A -85,B 0,C 180,E1 -3060.72,E2 -3060.72} C_VEL
LIN {X 0,Y 559.232,Z 275.452,A -85,B 0,C 180,E1 -3062.881,E2 -3062.881} C_VEL
LIN {X 0,Y 559.217,Z 275.452,A -85,B 0,C 180,E1 -3065.77,E2 -3065.77} C_VEL
LIN {X 0,Y 559.179,Z 275.455,A -85,B 0,C 180,E1 -3068.675,E2 -3068.675} C_VEL
LIN {X 0,Y 559.196,Z 275.452,A -85,B 0,C 180,E1 -3071.601,E2 -3071.601} C_VEL
LIN {X 0,Y 559.171,Z 275.455,A -85,B 0,C 180,E1 -3074.588,E2 -3074.588} C_VEL
LIN {X 0,Y 559.156,Z 275.457,A -85,B 0,C 180,E1 -3077.557,E2 -3077.557} C_VEL
LIN {X 0,Y 559.161,Z 275.462,A -85,B 0,C 180,E1 -3079.838,E2 -3079.838} C_VEL
LIN {X 0,Y 559.132,Z 275.461,A -85,B 0,C 180,E1 -3082.153,E2 -3082.153} C_VEL
LIN {X 0,Y 559.172,Z 275.456,A -85,B 0,C 180,E1 -3085.188,E2 -3085.188} C_VEL
LIN {X 0,Y 559.137,Z 275.463,A -85,B 0,C 180,E1 -3087.715,E2 -3087.715} C_VEL
LIN {X 0,Y 559.138,Z 275.459,A -85,B 0,C 180,E1 -3090.601,E2 -3090.601} C_VEL
LIN {X 0,Y 558.478,Z 275.543,A -85,B 0,C 180,E1 -3091.203,E2 -3091.203} C_VEL
LIN {X 0,Y 555.617,Z 275.903,A -85,B 0,C 180,E1 -3092.179,E2 -3092.179} C_VEL
LIN {X 0,Y 553.203,Z 276.2,A -85,B 0,C 180,E1 -3092.964,E2 -3092.964} C_VEL
LIN {X 0,Y 552.178,Z 276.331,A -85,B 0,C 180,E1 -3093.571,E2 -3093.571} C_VEL
LIN {X 0,Y 552.102,Z 276.335,A -85,B 0,C 180,E1 -3093.776,E2 -3093.776} C_VEL
LIN {X 0,Y 552.096,Z 276.343,A -85,B 0,C 180,E1 -3096.748,E2 -3096.748} C_VEL
LIN {X 0,Y 552.128,Z 276.336,A -85,B 0,C 180,E1 -3099.528,E2 -3099.528} C_VEL
LIN {X 0,Y 552.124,Z 276.336,A -85,B 0,C 180,E1 -3102.426,E2 -3102.426} C_VEL
LIN {X 0,Y 552.095,Z 276.34,A -85,B 0,C 180,E1 -3105.564,E2 -3105.564} C_VEL
LIN {X 0,Y 552.103,Z 276.341,A -85,B 0,C 180,E1 -3107.588,E2 -3107.588} C_VEL
LIN {X 0,Y 552.173,Z 277.316,A -85,B 0,C 180,E1 -3108.673,E2 -3108.673} C_VEL
LIN {X 0,Y 552.166,Z 281.614,A -85,B 0,C 180,E1 -3111.416,E2 -3111.416} C_VEL
LIN {X 0,Y 552.131,Z 286.076,A -85,B 0,C 180,E1 -3114.161,E2 -3114.161} C_VEL
LIN {X 0,Y 552.067,Z 291.126,A -85,B 0,C 180,E1 -3117.162,E2 -3117.162} C_VEL
LIN {X 0,Y 551.982,Z 296.45,A -85,B 0,C 180,E1 -3120.228,E2 -3120.228} C_VEL
LIN {X 0,Y 551.927,Z 300.887,A -85,B 0,C 180,E1 -3122.716,E2 -3122.716} C_VEL
LIN {X 0,Y 551.888,Z 305.307,A -85,B 0,C 180,E1 -3125.151,E2 -3125.151} C_VEL
LIN {X 0,Y 551.792,Z 309.723,A -85,B 0,C 180,E1 -3127.537,E2 -3127.537} C_VEL
LIN {X 0,Y 551.801,Z 315.657,A -85,B 0,C 180,E1 -3130.662,E2 -3130.662} C_VEL
LIN {X 0,Y 551.778,Z 317.782,A -85,B 0,C 180,E1 -3131.745,E2 -3131.745} C_VEL
LIN {X 0,Y 554.427,Z 329.274,A -85,B 0,C 180,E1 -3132.032,E2 -3132.032} C_VEL
LIN {X 0,Y 554.254,Z 344.692,A -85,B 0,C 180,E1 -3132.42,E2 -3132.42} C_VEL
LIN {X 0,Y 553.944,Z 359.823,A -85,B 0,C 180,E1 -3132.958,E2 -3132.958} C_VEL
LIN {X 0,Y 553.636,Z 373.529,A -85,B 0,C 180,E1 -3133.594,E2 -3133.594} C_VEL
LIN {X 0,Y 553.365,Z 386.527,A -85,B 0,C 180,E1 -3134.343,E2 -3134.343} C_VEL
LIN {X 0,Y 553.036,Z 399.806,A -85,B 0,C 180,E1 -3135.277,E2 -3135.277} C_VEL
LIN {X 0,Y 552.723,Z 410.908,A -85,B 0,C 180,E1 -3136.208,E2 -3136.208} C_VEL
LIN {X 0,Y 552.488,Z 422.101,A -85,B 0,C 180,E1 -3137.325,E2 -3137.325} C_VEL
LIN {X 0,Y 552.198,Z 433.343,A -85,B 0,C 180,E1 -3138.673,E2 -3138.673} C_VEL
LIN {X 0,Y 552.075,Z 442.014,A -85,B 0,C 180,E1 -3139.919,E2 -3139.919} C_VEL
LIN {X 0,Y 551.92,Z 449.503,A -85,B 0,C 180,E1 -3141.211,E2 -3141.211} C_VEL
LIN {X 0,Y 551.82,Z 456.506,A -85,B 0,C 180,E1 -3142.683,E2 -3142.683} C_VEL
LIN {X 0,Y 551.796,Z 462.014,A -85,B 0,C 180,E1 -3144.152,E2 -3144.152} C_VEL
LIN {X 0,Y 551.706,Z 466.181,A -85,B 0,C 180,E1 -3145.617,E2 -3145.617} C_VEL
LIN {X 0,Y 551.717,Z 469.114,A -85,B 0,C 180,E1 -3147.08,E2 -3147.08} C_VEL
LIN {X 0,Y 551.641,Z 470.879,A -85,B 0,C 180,E1 -3148.54,E2 -3148.54} C_VEL
LIN {X 0,Y 551.638,Z 471.496,A -85,B 0,C 180,E1 -3150,E2 -3150} C_VEL
LIN {X 0,Y 551.643,Z 470.94,A -85,B 0,C 180,E1 -3151.46,E2 -3151.46} C_VEL
LIN {X 0,Y 551.719,Z 469.255,A -85,B 0,C 180,E1 -3152.921,E2 -3152.921} C_VEL
LIN {X 0,Y 551.706,Z 466.401,A -85,B 0,C 180,E1 -3154.384,E2 -3154.384} C_VEL
LIN {X 0,Y 551.787,Z 462.313,A -85,B 0,C 180,E1 -3155.848,E2 -3155.848} C_VEL
LIN {X 0,Y 551.821,Z 456.897,A -85,B 0,C 180,E1 -3157.317,E2 -3157.317} C_VEL
LIN {X 0,Y 551.919,Z 449.995,A -85,B 0,C 180,E1 -3158.79,E2 -3158.79} C_VEL
LIN {X 0,Y 552.071,Z 442.567,A -85,B 0,C 180,E1 -3160.081,E2 -3160.081} C_VEL
LIN {X 0,Y 552.184,Z 434.058,A -85,B 0,C 180,E1 -3161.32,E2 -3161.32} C_VEL
LIN {X 0,Y 552.395,Z 424.53,A -85,B 0,C 180,E1 -3162.491,E2 -3162.491} C_VEL
LIN {X 0,Y 552.673,Z 413.798,A -85,B 0,C 180,E1 -3163.607,E2 -3163.607} C_VEL
LIN {X 0,Y 552.968,Z 402.086,A -85,B 0,C 180,E1 -3164.632,E2 -3164.632} C_VEL
LIN {X 0,Y 553.272,Z 389.301,A -85,B 0,C 180,E1 -3165.566,E2 -3165.566} C_VEL
LIN {X 0,Y 553.604,Z 375.202,A -85,B 0,C 180,E1 -3166.407,E2 -3166.407} C_VEL
LIN {X 0,Y 553.923,Z 360.746,A -85,B 0,C 180,E1 -3167.093,E2 -3167.093} C_VEL
LIN {X 0,Y 554.21,Z 345.208,A -85,B 0,C 180,E1 -3167.655,E2 -3167.655} C_VEL
LIN {X 0,Y 554.424,Z 329.877,A -85,B 0,C 180,E1 -3168.046,E2 -3168.046} C_VEL
LIN {X 0,Y 553.612,Z 325.31,A -85,B 0,C 180,E1 -3168.165,E2 -3168.165} C_VEL
LIN {X 0,Y 551.751,Z 317.727,A -85,B 0,C 180,E1 -3168.36,E2 -3168.36} C_VEL
LIN {X 0,Y 551.76,Z 312.845,A -85,B 0,C 180,E1 -3170.894,E2 -3170.894} C_VEL
LIN {X 0,Y 551.842,Z 307.917,A -85,B 0,C 180,E1 -3173.514,E2 -3173.514} C_VEL
LIN {X 0,Y 551.883,Z 303.969,A -85,B 0,C 180,E1 -3175.656,E2 -3175.656} C_VEL
LIN {X 0,Y 551.986,Z 298.791,A -85,B 0,C 180,E1 -3178.535,E2 -3178.535} C_VEL
LIN {X 0,Y 552.027,Z 293.65,A -85,B 0,C 180,E1 -3181.465,E2 -3181.465} C_VEL
LIN {X 0,Y 552.107,Z 289.021,A -85,B 0,C 180,E1 -3184.166,E2 -3184.166} C_VEL
LIN {X 0,Y 552.17,Z 284.737,A -85,B 0,C 180,E1 -3186.742,E2 -3186.742} C_VEL
LIN {X 0,Y 552.193,Z 280.268,A -85,B 0,C 180,E1 -3189.521,E2 -3189.521} C_VEL
LIN {X 0,Y 552.164,Z 277.282,A -85,B 0,C 180,E1 -3191.442,E2 -3191.442} C_VEL
LIN {X 0,Y 552.107,Z 276.341,A -85,B 0,C 180,E1 -3192.427,E2 -3192.427} C_VEL
LIN {X 0,Y 552.097,Z 276.343,A -85,B 0,C 180,E1 -3195.562,E2 -3195.562} C_VEL
LIN {X 0,Y 552.117,Z 276.338,A -85,B 0,C 180,E1 -3198.554,E2 -3198.554} C_VEL
LIN {X 0,Y 552.119,Z 276.336,A -85,B 0,C 180,E1 -3201.411,E2 -3201.411} C_VEL
LIN {X 0,Y 552.072,Z 276.341,A -85,B 0,C 180,E1 -3204.155,E2 -3204.155} C_VEL
LIN {X 0,Y 552.113,Z 276.337,A -85,B 0,C 180,E1 -3206.814,E2 -3206.814} C_VEL
LIN {X 0,Y 552.104,Z 276.341,A -85,B 0,C 180,E1 -3209.391,E2 -3209.391} C_VEL
LIN {X 0,Y 552.074,Z 276.34,A -85,B 0,C 180,E1 -3211.9,E2 -3211.9} C_VEL
LIN {X 0,Y 552.134,Z 276.333,A -85,B 0,C 180,E1 -3214.653,E2 -3214.653} C_VEL
LIN {X 0,Y 552.091,Z 276.338,A -85,B 0,C 180,E1 -3217.549,E2 -3217.549} C_VEL
LIN {X 0,Y 552.147,Z 276.331,A -85,B 0,C 180,E1 -3220.674,E2 -3220.674} C_VEL
LIN {X 0,Y 552.111,Z 276.335,A -85,B 0,C 180,E1 -3223.737,E2 -3223.737} C_VEL
LIN {X 0,Y 552.114,Z 276.337,A -85,B 0,C 180,E1 -3226.004,E2 -3226.004} C_VEL
LIN {X 0,Y 552.16,Z 276.331,A -85,B 0,C 180,E1 -3228.993,E2 -3228.993} C_VEL
LIN {X 0,Y 552.15,Z 276.331,A -85,B 0,C 180,E1 -3231.951,E2 -3231.951} C_VEL
LIN {X 0,Y 552.224,Z 276.322,A -85,B 0,C 180,E1 -3234.889,E2 -3234.889} C_VEL
LIN {X 0,Y 552.224,Z 276.321,A -85,B 0,C 180,E1 -3237.812,E2 -3237.812} C_VEL
LIN {X 0,Y 552.228,Z 276.321,A -85,B 0,C 180,E1 -3240.729,E2 -3240.729} C_VEL
LIN {X 0,Y 552.201,Z 276.328,A -85,B 0,C 180,E1 -3242.918,E2 -3242.918} C_VEL
LIN {X 0,Y 552.188,Z 276.328,A -85,B 0,C 180,E1 -3245.844,E2 -3245.844} C_VEL
LIN {X 0,Y 552.153,Z 276.331,A -85,B 0,C 180,E1 -3248.786,E2 -3248.786} C_VEL
LIN {X 0,Y 552.158,Z 276.33,A -85,B 0,C 180,E1 -3251.751,E2 -3251.751} C_VEL
LIN {X 0,Y 552.124,Z 276.334,A -85,B 0,C 180,E1 -3254.749,E2 -3254.749} C_VEL
LIN {X 0,Y 552.11,Z 276.336,A -85,B 0,C 180,E1 -3257.788,E2 -3257.788} C_VEL
LIN {X 0,Y 552.12,Z 276.338,A -85,B 0,C 180,E1 -3260.102,E2 -3260.102} C_VEL
LIN {X 0,Y 552.086,Z 276.339,A -85,B 0,C 180,E1 -3262.451,E2 -3262.451} C_VEL
LIN {X 0,Y 552.152,Z 276.33,A -85,B 0,C 180,E1 -3265.351,E2 -3265.351} C_VEL
LIN {X 0,Y 552.083,Z 276.34,A -85,B 0,C 180,E1 -3268.1,E2 -3268.1} C_VEL
LIN {X 0,Y 552.099,Z 276.343,A -85,B 0,C 180,E1 -3270.609,E2 -3270.609} C_VEL
LIN {X 0,Y 552.112,Z 276.338,A -85,B 0,C 180,E1 -3273.186,E2 -3273.186} C_VEL
LIN {X 0,Y 552.07,Z 276.342,A -85,B 0,C 180,E1 -3275.845,E2 -3275.845} C_VEL
LIN {X 0,Y 552.118,Z 276.338,A -85,B 0,C 180,E1 -3278.589,E2 -3278.589} C_VEL
LIN {X 0,Y 552.114,Z 276.34,A -85,B 0,C 180,E1 -3281.446,E2 -3281.446} C_VEL
LIN {X 0,Y 552.093,Z 276.344,A -85,B 0,C 180,E1 -3284.532,E2 -3284.532} C_VEL
LIN {X 0,Y 552.132,Z 276.386,A -85,B 0,C 180,E1 -3287.452,E2 -3287.452} C_VEL
LIN {X 0,Y 552.414,Z 280.13,A -85,B 0,C 180,E1 -3289.546,E2 -3289.546} C_VEL
LIN {X 0,Y 552.304,Z 285.452,A -85,B 0,C 180,E1 -3292.353,E2 -3292.353} C_VEL
LIN {X 0,Y 552.221,Z 290.776,A -85,B 0,C 180,E1 -3295.061,E2 -3295.061} C_VEL
LIN {X 0,Y 552.151,Z 296.114,A -85,B 0,C 180,E1 -3297.684,E2 -3297.684} C_VEL
LIN {X 0,Y 552.063,Z 301.486,A -85,B 0,C 180,E1 -3300.232,E2 -3300.232} C_VEL
LIN {X 0,Y 551.996,Z 307.53,A -85,B 0,C 180,E1 -3303.029,E2 -3303.029} C_VEL
LIN {X 0,Y 551.889,Z 314.005,A -85,B 0,C 180,E1 -3305.952,E2 -3305.952} C_VEL
LIN {X 0,Y 551.911,Z 319.454,A -85,B 0,C 180,E1 -3308.369,E2 -3308.369} C_VEL
LIN {X 0,Y 551.806,Z 326.457,A -85,B 0,C 180,E1 -3311.433,E2 -3311.433} C_VEL
LIN {X 0,Y 551.829,Z 327.049,A -85,B 0,C 180,E1 -3311.691,E2 -3311.691} C_VEL
LIN {X 0,Y 554.427,Z 338.415,A -85,B 0,C 180,E1 -3311.969,E2 -3311.969} C_VEL
LIN {X 0,Y 554.211,Z 353.413,A -85,B 0,C 180,E1 -3312.334,E2 -3312.334} C_VEL
LIN {X 0,Y 553.936,Z 368.795,A -85,B 0,C 180,E1 -3312.87,E2 -3312.87} C_VEL
LIN {X 0,Y 553.658,Z 382.598,A -85,B 0,C 180,E1 -3313.5,E2 -3313.5} C_VEL
LIN {X 0,Y 553.358,Z 395.773,A -85,B 0,C 180,E1 -3314.248,E2 -3314.248} C_VEL
LIN {X 0,Y 553.054,Z 409.299,A -85,B 0,C 180,E1 -3315.192,E2 -3315.192} C_VEL
LIN {X 0,Y 552.712,Z 421.378,A -85,B 0,C 180,E1 -3316.207,E2 -3316.207} C_VEL
LIN {X 0,Y 552.482,Z 432.508,A -85,B 0,C 180,E1 -3317.324,E2 -3317.324} C_VEL
LIN {X 0,Y 552.216,Z 442.484,A -85,B 0,C 180,E1 -3318.513,E2 -3318.513} C_VEL
LIN {X 0,Y 552.124,Z 451.086,A -85,B 0,C 180,E1 -3319.735,E2 -3319.735} C_VEL
LIN {X 0,Y 551.921,Z 458.742,A -85,B 0,C 180,E1 -3321.026,E2 -3321.026} C_VEL
LIN {X 0,Y 551.837,Z 465.089,A -85,B 0,C 180,E1 -3322.315,E2 -3322.315} C_VEL
LIN {X 0,Y 551.769,Z 470.57,A -85,B 0,C 180,E1 -3323.68,E2 -3323.68} C_VEL
LIN {X 0,Y 551.713,Z 474.386,A -85,B 0,C 180,E1 -3324.884,E2 -3324.884} C_VEL
LIN {X 0,Y 551.73,Z 477.888,A -85,B 0,C 180,E1 -3326.348,E2 -3326.348} C_VEL
LIN {X 0,Y 551.655,Z 480.191,A -85,B 0,C 180,E1 -3327.809,E2 -3327.809} C_VEL
LIN {X 0,Y 551.637,Z 481.348,A -85,B 0,C 180,E1 -3329.27,E2 -3329.27} C_VEL
LIN {X 0,Y 551.637,Z 481.348,A -85,B 0,C 180,E1 -3330.73,E2 -3330.73} C_VEL
LIN {X 0,Y 551.655,Z 480.189,A -85,B 0,C 180,E1 -3332.19,E2 -3332.19} C_VEL
LIN {X 0,Y 551.73,Z 477.886,A -85,B 0,C 180,E1 -3333.651,E2 -3333.651} C_VEL
LIN {X 0,Y 551.713,Z 474.387,A -85,B 0,C 180,E1 -3335.115,E2 -3335.115} C_VEL
LIN {X 0,Y 551.82,Z 469.61,A -85,B 0,C 180,E1 -3336.582,E2 -3336.582} C_VEL
LIN {X 0,Y 551.876,Z 463.424,A -85,B 0,C 180,E1 -3338.052,E2 -3338.052} C_VEL
LIN {X 0,Y 551.95,Z 455.648,A -85,B 0,C 180,E1 -3339.528,E2 -3339.528} C_VEL
LIN {X 0,Y 552.183,Z 447.371,A -85,B 0,C 180,E1 -3340.82,E2 -3340.82} C_VEL
LIN {X 0,Y 552.352,Z 437.395,A -85,B 0,C 180,E1 -3342.118,E2 -3342.118} C_VEL
LIN {X 0,Y 552.608,Z 427.191,A -85,B 0,C 180,E1 -3343.233,E2 -3343.233} C_VEL
LIN {X 0,Y 552.906,Z 415.025,A -85,B 0,C 180,E1 -3344.351,E2 -3344.351} C_VEL
LIN {X 0,Y 553.224,Z 402.451,A -85,B 0,C 180,E1 -3345.31,E2 -3345.31} C_VEL
LIN {X 0,Y 553.483,Z 389.518,A -85,B 0,C 180,E1 -3346.126,E2 -3346.126} C_VEL
LIN {X 0,Y 553.813,Z 374.837,A -85,B 0,C 180,E1 -3346.875,E2 -3346.875} C_VEL
LIN {X 0,Y 554.141,Z 360.181,A -85,B 0,C 180,E1 -3347.451,E2 -3347.451} C_VEL
LIN {X 0,Y 554.343,Z 344.984,A -85,B 0,C 180,E1 -3347.891,E2 -3347.891} C_VEL
LIN {X 0,Y 554.25,Z 337.077,A -85,B 0,C 180,E1 -3348.065,E2 -3348.065} C_VEL
LIN {X 0,Y 551.824,Z 327.036,A -85,B 0,C 180,E1 -3348.315,E2 -3348.315} C_VEL
LIN {X 0,Y 551.845,Z 321.14,A -85,B 0,C 180,E1 -3350.89,E2 -3350.89} C_VEL
LIN {X 0,Y 551.885,Z 315.165,A -85,B 0,C 180,E1 -3353.525,E2 -3353.525} C_VEL
LIN {X 0,Y 551.944,Z 310.408,A -85,B 0,C 180,E1 -3355.653,E2 -3355.653} C_VEL
LIN {X 0,Y 552.068,Z 304.063,A -85,B 0,C 180,E1 -3358.551,E2 -3358.551} C_VEL
LIN {X 0,Y 552.107,Z 297.869,A -85,B 0,C 180,E1 -3361.475,E2 -3361.475} C_VEL
LIN {X 0,Y 552.211,Z 292.3,A -85,B 0,C 180,E1 -3364.182,E2 -3364.182} C_VEL
LIN {X 0,Y 552.294,Z 287.229,A -85,B 0,C 180,E1 -3366.731,E2 -3366.731} C_VEL
LIN {X 0,Y 552.349,Z 281.908,A -85,B 0,C 180,E1 -3369.507,E2 -3369.507} C_VEL
LIN {X 0,Y 552.375,Z 278.364,A -85,B 0,C 180,E1 -3371.422,E2 -3371.422} C_VEL
LIN {X 0,Y 552.122,Z 276.339,A -85,B 0,C 180,E1 -3372.672,E2 -3372.672} C_VEL
LIN {X 0,Y 552.092,Z 276.343,A -85,B 0,C 180,E1 -3375.562,E2 -3375.562} C_VEL
LIN {X 0,Y 552.125,Z 276.34,A -85,B 0,C 180,E1 -3378.677,E2 -3378.677} C_VEL
LIN {X 0,Y 552.115,Z 276.337,A -85,B 0,C 180,E1 -3381.411,E2 -3381.411} C_VEL
LIN {X 0,Y 552.067,Z 276.342,A -85,B 0,C 180,E1 -3384.155,E2 -3384.155} C_VEL
LIN {X 0,Y 552.114,Z 276.337,A -85,B 0,C 180,E1 -3386.814,E2 -3386.814} C_VEL
LIN {X 0,Y 552.1,Z 276.344,A -85,B 0,C 180,E1 -3389.391,E2 -3389.391} C_VEL
LIN {X 0,Y 552.083,Z 276.34,A -85,B 0,C 180,E1 -3391.9,E2 -3391.9} C_VEL
LIN {X 0,Y 552.147,Z 276.331,A -85,B 0,C 180,E1 -3394.649,E2 -3394.649} C_VEL
LIN {X 0,Y 552.086,Z 276.339,A -85,B 0,C 180,E1 -3397.549,E2 -3397.549} C_VEL
LIN {X 0,Y 552.148,Z 276.331,A -85,B 0,C 180,E1 -3400.674,E2 -3400.674} C_VEL
LIN {X 0,Y 552.106,Z 276.336,A -85,B 0,C 180,E1 -3403.737,E2 -3403.737} C_VEL
LIN {X 0,Y 552.119,Z 276.337,A -85,B 0,C 180,E1 -3406.004,E2 -3406.004} C_VEL
LIN {X 0,Y 552.171,Z 276.33,A -85,B 0,C 180,E1 -3408.994,E2 -3408.994} C_VEL
LIN {X 0,Y 552.145,Z 276.332,A -85,B 0,C 180,E1 -3411.951,E2 -3411.951} C_VEL
LIN {X 0,Y 552.223,Z 276.321,A -85,B 0,C 180,E1 -3414.889,E2 -3414.889} C_VEL
LIN {X 0,Y 552.221,Z 276.32,A -85,B 0,C 180,E1 -3417.812,E2 -3417.812} C_VEL
LIN {X 0,Y 552.225,Z 276.321,A -85,B 0,C 180,E1 -3420.729,E2 -3420.729} C_VEL
LIN {X 0,Y 552.199,Z 276.328,A -85,B 0,C 180,E1 -3422.918,E2 -3422.918} C_VEL
LIN {X 0,Y 552.185,Z 276.328,A -85,B 0,C 180,E1 -3425.844,E2 -3425.844} C_VEL
LIN {X 0,Y 552.151,Z 276.331,A -85,B 0,C 180,E1 -3428.786,E2 -3428.786} C_VEL
LIN {X 0,Y 552.153,Z 276.33,A -85,B 0,C 180,E1 -3431.751,E2 -3431.751} C_VEL
LIN {X 0,Y 552.119,Z 276.334,A -85,B 0,C 180,E1 -3434.749,E2 -3434.749} C_VEL
LIN {X 0,Y 552.107,Z 276.335,A -85,B 0,C 180,E1 -3437.789,E2 -3437.789} C_VEL
LIN {X 0,Y 552.12,Z 276.337,A -85,B 0,C 180,E1 -3440.102,E2 -3440.102} C_VEL
LIN {X 0,Y 552.087,Z 276.339,A -85,B 0,C 180,E1 -3442.451,E2 -3442.451} C_VEL
LIN {X 0,Y 552.148,Z 276.331,A -85,B 0,C 180,E1 -3445.351,E2 -3445.351} C_VEL
LIN {X 0,Y 552.083,Z 276.338,A -85,B 0,C 180,E1 -3448.1,E2 -3448.1} C_VEL
LIN {X 0,Y 552.1,Z 276.341,A -85,B 0,C 180,E1 -3450.609,E2 -3450.609} C_VEL
LIN {X 0,Y 552.114,Z 276.335,A -85,B 0,C 180,E1 -3453.186,E2 -3453.186} C_VEL
LIN {X 0,Y 552.102,Z 276.335,A -85,B 0,C 180,E1 -3453.776,E2 -3453.776} C_VEL
LIN {X 0,Y 551.462,Z 276.418,A -85,B 0,C 180,E1 -3454.385,E2 -3454.385} C_VEL
LIN {X 0,Y 548.639,Z 276.775,A -85,B 0,C 180,E1 -3455.373,E2 -3455.373} C_VEL
LIN {X 0,Y 546.222,Z 277.077,A -85,B 0,C 180,E1 -3456.168,E2 -3456.168} C_VEL
LIN {X 0,Y 545.156,Z 277.207,A -85,B 0,C 180,E1 -3456.782,E2 -3456.782} C_VEL
LIN {X 0,Y 545.055,Z 277.217,A -85,B 0,C 180,E1 -3456.99,E2 -3456.99} C_VEL
LIN {X 0,Y 545.066,Z 277.215,A -85,B 0,C 180,E1 -3460.143,E2 -3460.143} C_VEL
LIN {X 0,Y 545.073,Z 277.215,A -85,B 0,C 180,E1 -3463.107,E2 -3463.107} C_VEL
LIN {X 0,Y 545.06,Z 277.218,A -85,B 0,C 180,E1 -3466.225,E2 -3466.225} C_VEL
LIN {X 0,Y 545.036,Z 277.222,A -85,B 0,C 180,E1 -3467.894,E2 -3467.894} C_VEL
LIN {X 0,Y 545.166,Z 280.163,A -85,B 0,C 180,E1 -3469.867,E2 -3469.867} C_VEL
LIN {X 0,Y 545.123,Z 285.206,A -85,B 0,C 180,E1 -3473.067,E2 -3473.067} C_VEL
LIN {X 0,Y 545.063,Z 289.369,A -85,B 0,C 180,E1 -3475.61,E2 -3475.61} C_VEL
LIN {X 0,Y 544.971,Z 293.965,A -85,B 0,C 180,E1 -3478.336,E2 -3478.336} C_VEL
LIN {X 0,Y 544.939,Z 299.447,A -85,B 0,C 180,E1 -3481.499,E2 -3481.499} C_VEL
LIN {X 0,Y 544.853,Z 305.356,A -85,B 0,C 180,E1 -3484.808,E2 -3484.808} C_VEL
LIN {X 0,Y 544.724,Z 309.772,A -85,B 0,C 180,E1 -3487.229,E2 -3487.229} C_VEL
LIN {X 0,Y 544.733,Z 315.669,A -85,B 0,C 180,E1 -3490.401,E2 -3490.401} C_VEL
LIN {X 0,Y 544.671,Z 317.738,A -85,B 0,C 180,E1 -3491.489,E2 -3491.489} C_VEL
LIN {X 0,Y 547.669,Z 330.582,A -85,B 0,C 180,E1 -3491.829,E2 -3491.829} C_VEL
LIN {X 0,Y 547.464,Z 345.708,A -85,B 0,C 180,E1 -3492.227,E2 -3492.227} C_VEL
LIN {X 0,Y 547.134,Z 359.943,A -85,B 0,C 180,E1 -3492.744,E2 -3492.744} C_VEL
LIN {X 0,Y 546.802,Z 373.538,A -85,B 0,C 180,E1 -3493.383,E2 -3493.383} C_VEL
LIN {X 0,Y 546.473,Z 386.533,A -85,B 0,C 180,E1 -3494.14,E2 -3494.14} C_VEL
LIN {X 0,Y 546.116,Z 399.811,A -85,B 0,C 180,E1 -3495.086,E2 -3495.086} C_VEL
LIN {X 0,Y 545.786,Z 410.915,A -85,B 0,C 180,E1 -3496.029,E2 -3496.029} C_VEL
LIN {X 0,Y 545.525,Z 422.106,A -85,B 0,C 180,E1 -3497.16,E2 -3497.16} C_VEL
LIN {X 0,Y 545.204,Z 432.661,A -85,B 0,C 180,E1 -3498.431,E2 -3498.431} C_VEL
LIN {X 0,Y 545.05,Z 442.017,A -85,B 0,C 180,E1 -3499.788,E2 -3499.788} C_VEL
LIN {X 0,Y 544.846,Z 449.505,A -85,B 0,C 180,E1 -3501.096,E2 -3501.096} C_VEL
LIN {X 0,Y 544.746,Z 456.508,A -85,B 0,C 180,E1 -3502.588,E2 -3502.588} C_VEL
LIN {X 0,Y 544.708,Z 462.016,A -85,B 0,C 180,E1 -3504.076,E2 -3504.076} C_VEL
LIN {X 0,Y 544.605,Z 466.182,A -85,B 0,C 180,E1 -3505.56,E2 -3505.56} C_VEL
LIN {X 0,Y 544.643,Z 469.114,A -85,B 0,C 180,E1 -3507.042,E2 -3507.042} C_VEL
LIN {X 0,Y 544.543,Z 470.879,A -85,B 0,C 180,E1 -3508.521,E2 -3508.521} C_VEL
LIN {X 0,Y 544.539,Z 471.496,A -85,B 0,C 180,E1 -3510,E2 -3510} C_VEL
LIN {X 0,Y 544.544,Z 470.939,A -85,B 0,C 180,E1 -3511.479,E2 -3511.479} C_VEL
LIN {X 0,Y 544.645,Z 469.253,A -85,B 0,C 180,E1 -3512.959,E2 -3512.959} C_VEL
LIN {X 0,Y 544.605,Z 466.4,A -85,B 0,C 180,E1 -3514.441,E2 -3514.441} C_VEL
LIN {X 0,Y 544.696,Z 462.312,A -85,B 0,C 180,E1 -3515.925,E2 -3515.925} C_VEL
LIN {X 0,Y 544.746,Z 456.894,A -85,B 0,C 180,E1 -3517.413,E2 -3517.413} C_VEL
LIN {X 0,Y 544.846,Z 449.992,A -85,B 0,C 180,E1 -3518.905,E2 -3518.905} C_VEL
LIN {X 0,Y 545.081,Z 441.38,A -85,B 0,C 180,E1 -3520.4,E2 -3520.4} C_VEL
LIN {X 0,Y 545.232,Z 431.751,A -85,B 0,C 180,E1 -3521.774,E2 -3521.774} C_VEL
LIN {X 0,Y 545.53,Z 421.171,A -85,B 0,C 180,E1 -3523.029,E2 -3523.029} C_VEL
LIN {X 0,Y 545.83,Z 409.795,A -85,B 0,C 180,E1 -3524.161,E2 -3524.161} C_VEL
LIN {X 0,Y 546.148,Z 397.6,A -85,B 0,C 180,E1 -3525.176,E2 -3525.176} C_VEL
LIN {X 0,Y 546.547,Z 384.986,A -85,B 0,C 180,E1 -3526.049,E2 -3526.049} C_VEL
LIN {X 0,Y 546.863,Z 371.656,A -85,B 0,C 180,E1 -3526.808,E2 -3526.808} C_VEL
LIN {X 0,Y 547.212,Z 358.011,A -85,B 0,C 180,E1 -3527.425,E2 -3527.425} C_VEL
LIN {X 0,Y 547.492,Z 343.131,A -85,B 0,C 180,E1 -3527.944,E2 -3527.944} C_VEL
LIN {X 0,Y 547.529,Z 329.281,A -85,B 0,C 180,E1 -3528.293,E2 -3528.293} C_VEL
LIN {X 0,Y 544.664,Z 317.722,A -85,B 0,C 180,E1 -3528.609,E2 -3528.609} C_VEL
LIN {X 0,Y 544.688,Z 312.874,A -85,B 0,C 180,E1 -3531.179,E2 -3531.179} C_VEL
LIN {X 0,Y 544.79,Z 308.273,A -85,B 0,C 180,E1 -3533.662,E2 -3533.662} C_VEL
LIN {X 0,Y 544.798,Z 304.028,A -85,B 0,C 180,E1 -3536.015,E2 -3536.015} C_VEL
LIN {X 0,Y 544.93,Z 299.254,A -85,B 0,C 180,E1 -3538.717,E2 -3538.717} C_VEL
LIN {X 0,Y 544.968,Z 293.686,A -85,B 0,C 180,E1 -3541.92,E2 -3541.92} C_VEL
LIN {X 0,Y 545.063,Z 289.23,A -85,B 0,C 180,E1 -3544.564,E2 -3544.564} C_VEL
LIN {X 0,Y 545.127,Z 284.767,A -85,B 0,C 180,E1 -3547.296,E2 -3547.296} C_VEL
LIN {X 0,Y 545.184,Z 279.75,A -85,B 0,C 180,E1 -3550.485,E2 -3550.485} C_VEL
LIN {X 0,Y 545.04,Z 277.305,A -85,B 0,C 180,E1 -3552.106,E2 -3552.106} C_VEL
LIN {X 0,Y 545.061,Z 277.216,A -85,B 0,C 180,E1 -3555.167,E2 -3555.167} C_VEL
LIN {X 0,Y 545.075,Z 277.212,A -85,B 0,C 180,E1 -3557.897,E2 -3557.897} C_VEL
LIN {X 0,Y 545.083,Z 277.212,A -85,B 0,C 180,E1 -3560.818,E2 -3560.818} C_VEL
LIN {X 0,Y 545.034,Z 277.22,A -85,B 0,C 180,E1 -3563.619,E2 -3563.619} C_VEL
LIN {X 0,Y 545.061,Z 277.219,A -85,B 0,C 180,E1 -3566.328,E2 -3566.328} C_VEL
LIN {X 0,Y 545.065,Z 277.214,A -85,B 0,C 180,E1 -3568.952,E2 -3568.952} C_VEL
LIN {X 0,Y 545.072,Z 277.213,A -85,B 0,C 180,E1 -3571.506,E2 -3571.506} C_VEL
LIN {X 0,Y 545.081,Z 277.212,A -85,B 0,C 180,E1 -3574.493,E2 -3574.493} C_VEL
LIN {X 0,Y 545.041,Z 277.219,A -85,B 0,C 180,E1 -3577.242,E2 -3577.242} C_VEL
LIN {X 0,Y 545.112,Z 277.209,A -85,B 0,C 180,E1 -3580.414,E2 -3580.414} C_VEL
LIN {X 0,Y 545.068,Z 277.214,A -85,B 0,C 180,E1 -3583.521,E2 -3583.521} C_VEL
LIN {X 0,Y 545.077,Z 277.212,A -85,B 0,C 180,E1 -3585.819,E2 -3585.819} C_VEL
LIN {X 0,Y 545.115,Z 277.207,A -85,B 0,C 180,E1 -3588.849,E2 -3588.849} C_VEL
LIN {X 0,Y 545.122,Z 277.206,A -85,B 0,C 180,E1 -3591.847,E2 -3591.847} C_VEL
LIN {X 0,Y 545.199,Z 277.196,A -85,B 0,C 180,E1 -3594.823,E2 -3594.823} C_VEL
LIN {X 0,Y 545.195,Z 277.197,A -85,B 0,C 180,E1 -3597.784,E2 -3597.784} C_VEL
LIN {X 0,Y 545.199,Z 277.196,A -85,B 0,C 180,E1 -3600.739,E2 -3600.739} C_VEL
LIN {X 0,Y 545.169,Z 277.204,A -85,B 0,C 180,E1 -3602.956,E2 -3602.956} C_VEL
LIN {X 0,Y 545.157,Z 277.204,A -85,B 0,C 180,E1 -3605.92,E2 -3605.92} C_VEL
LIN {X 0,Y 545.113,Z 277.209,A -85,B 0,C 180,E1 -3608.9,E2 -3608.9} C_VEL
LIN {X 0,Y 545.13,Z 277.207,A -85,B 0,C 180,E1 -3611.904,E2 -3611.904} C_VEL
LIN {X 0,Y 545.077,Z 277.213,A -85,B 0,C 180,E1 -3614.944,E2 -3614.944} C_VEL
LIN {X 0,Y 545.077,Z 277.213,A -85,B 0,C 180,E1 -3618.026,E2 -3618.026} C_VEL
LIN {X 0,Y 545.086,Z 277.211,A -85,B 0,C 180,E1 -3620.372,E2 -3620.372} C_VEL
LIN {X 0,Y 545.077,Z 277.212,A -85,B 0,C 180,E1 -3623.559,E2 -3623.559} C_VEL
LIN {X 0,Y 545.074,Z 277.217,A -85,B 0,C 180,E1 -3626.001,E2 -3626.001} C_VEL
LIN {X 0,Y 545.067,Z 277.215,A -85,B 0,C 180,E1 -3628.745,E2 -3628.745} C_VEL
LIN {X 0,Y 545.054,Z 277.217,A -85,B 0,C 180,E1 -3631.679,E2 -3631.679} C_VEL
LIN {X 0,Y 545.054,Z 277.217,A -85,B 0,C 180,E1 -3634.565,E2 -3634.565} C_VEL
LIN {X 0,Y 545.033,Z 277.22,A -85,B 0,C 180,E1 -3637.304,E2 -3637.304} C_VEL
LIN {X 0,Y 545.066,Z 277.216,A -85,B 0,C 180,E1 -3640.143,E2 -3640.143} C_VEL
LIN {X 0,Y 545.042,Z 277.221,A -85,B 0,C 180,E1 -3643.11,E2 -3643.11} C_VEL
LIN {X 0,Y 545.057,Z 277.221,A -85,B 0,C 180,E1 -3645.871,E2 -3645.871} C_VEL
LIN {X 0,Y 545.089,Z 277.295,A -85,B 0,C 180,E1 -3647.3,E2 -3647.3} C_VEL
LIN {X 0,Y 545.413,Z 281.144,A -85,B 0,C 180,E1 -3649.486,E2 -3649.486} C_VEL
LIN {X 0,Y 545.261,Z 287.198,A -85,B 0,C 180,E1 -3652.714,E2 -3652.714} C_VEL
LIN {X 0,Y 545.173,Z 292.817,A -85,B 0,C 180,E1 -3655.593,E2 -3655.593} C_VEL
LIN {X 0,Y 545.064,Z 298.34,A -85,B 0,C 180,E1 -3658.32,E2 -3658.32} C_VEL
LIN {X 0,Y 545.014,Z 305.03,A -85,B 0,C 180,E1 -3661.503,E2 -3661.503} C_VEL
LIN {X 0,Y 544.871,Z 311.599,A -85,B 0,C 180,E1 -3664.541,E2 -3664.541} C_VEL
LIN {X 0,Y 544.813,Z 317.543,A -85,B 0,C 180,E1 -3667.232,E2 -3667.232} C_VEL
LIN {X 0,Y 544.772,Z 322.898,A -85,B 0,C 180,E1 -3669.615,E2 -3669.615} C_VEL
LIN {X 0,Y 544.741,Z 327.128,A -85,B 0,C 180,E1 -3671.446,E2 -3671.446} C_VEL
LIN {X 0,Y 547.68,Z 339.54,A -85,B 0,C 180,E1 -3671.763,E2 -3671.763} C_VEL
LIN {X 0,Y 547.409,Z 355.072,A -85,B 0,C 180,E1 -3672.16,E2 -3672.16} C_VEL
LIN {X 0,Y 547.142,Z 369.004,A -85,B 0,C 180,E1 -3672.66,E2 -3672.66} C_VEL
LIN {X 0,Y 546.825,Z 382.596,A -85,B 0,C 180,E1 -3673.287,E2 -3673.287} C_VEL
LIN {X 0,Y 546.488,Z 395.77,A -85,B 0,C 180,E1 -3674.045,E2 -3674.045} C_VEL
LIN {X 0,Y 546.17,Z 408.899,A -85,B 0,C 180,E1 -3674.969,E2 -3674.969} C_VEL
LIN {X 0,Y 545.776,Z 421.376,A -85,B 0,C 180,E1 -3676.028,E2 -3676.028} C_VEL
LIN {X 0,Y 545.511,Z 432.508,A -85,B 0,C 180,E1 -3677.159,E2 -3677.159} C_VEL
LIN {X 0,Y 545.175,Z 443.103,A -85,B 0,C 180,E1 -3678.446,E2 -3678.446} C_VEL
LIN {X 0,Y 545.05,Z 452.295,A -85,B 0,C 180,E1 -3679.788,E2 -3679.788} C_VEL
LIN {X 0,Y 544.845,Z 459.749,A -85,B 0,C 180,E1 -3681.095,E2 -3681.095} C_VEL
LIN {X 0,Y 544.745,Z 466.7,A -85,B 0,C 180,E1 -3682.587,E2 -3682.587} C_VEL
LIN {X 0,Y 544.709,Z 472.162,A -85,B 0,C 180,E1 -3684.075,E2 -3684.075} C_VEL
LIN {X 0,Y 544.606,Z 476.291,A -85,B 0,C 180,E1 -3685.559,E2 -3685.559} C_VEL
LIN {X 0,Y 544.643,Z 479.185,A -85,B 0,C 180,E1 -3687.041,E2 -3687.041} C_VEL
LIN {X 0,Y 544.543,Z 480.91,A -85,B 0,C 180,E1 -3688.521,E2 -3688.521} C_VEL
LIN {X 0,Y 544.538,Z 481.5,A -85,B 0,C 180,E1 -3690,E2 -3690} C_VEL
LIN {X 0,Y 544.543,Z 480.909,A -85,B 0,C 180,E1 -3691.479,E2 -3691.479} C_VEL
LIN {X 0,Y 544.643,Z 479.182,A -85,B 0,C 180,E1 -3692.958,E2 -3692.958} C_VEL
LIN {X 0,Y 544.606,Z 476.29,A -85,B 0,C 180,E1 -3694.44,E2 -3694.44} C_VEL
LIN {X 0,Y 544.709,Z 472.166,A -85,B 0,C 180,E1 -3695.924,E2 -3695.924} C_VEL
LIN {X 0,Y 544.744,Z 466.703,A -85,B 0,C 180,E1 -3697.412,E2 -3697.412} C_VEL
LIN {X 0,Y 544.845,Z 459.747,A -85,B 0,C 180,E1 -3698.904,E2 -3698.904} C_VEL
LIN {X 0,Y 545.073,Z 451.086,A -85,B 0,C 180,E1 -3700.399,E2 -3700.399} C_VEL
LIN {X 0,Y 545.236,Z 441.711,A -85,B 0,C 180,E1 -3701.734,E2 -3701.734} C_VEL
LIN {X 0,Y 545.51,Z 432.512,A -85,B 0,C 180,E1 -3702.84,E2 -3702.84} C_VEL
LIN {X 0,Y 545.827,Z 420.364,A -85,B 0,C 180,E1 -3704.065,E2 -3704.065} C_VEL
LIN {X 0,Y 546.191,Z 407.812,A -85,B 0,C 180,E1 -3705.115,E2 -3705.115} C_VEL
LIN {X 0,Y 546.54,Z 394.259,A -85,B 0,C 180,E1 -3706.049,E2 -3706.049} C_VEL
LIN {X 0,Y 546.868,Z 380.784,A -85,B 0,C 180,E1 -3706.807,E2 -3706.807} C_VEL
LIN {X 0,Y 547.246,Z 366.188,A -85,B 0,C 180,E1 -3707.455,E2 -3707.455} C_VEL
LIN {X 0,Y 547.536,Z 350.859,A -85,B 0,C 180,E1 -3707.966,E2 -3707.966} C_VEL
LIN {X 0,Y 547.519,Z 338.356,A -85,B 0,C 180,E1 -3708.268,E2 -3708.268} C_VEL
LIN {X 0,Y 544.742,Z 327.022,A -85,B 0,C 180,E1 -3708.568,E2 -3708.568} C_VEL
LIN {X 0,Y 544.794,Z 321.107,A -85,B 0,C 180,E1 -3711.174,E2 -3711.174} C_VEL
LIN {X 0,Y 544.83,Z 315.512,A -85,B 0,C 180,E1 -3713.672,E2 -3713.672} C_VEL
LIN {X 0,Y 544.895,Z 310.363,A -85,B 0,C 180,E1 -3716.009,E2 -3716.009} C_VEL
LIN {X 0,Y 544.999,Z 304.504,A -85,B 0,C 180,E1 -3718.731,E2 -3718.731} C_VEL
LIN {X 0,Y 545.07,Z 297.865,A -85,B 0,C 180,E1 -3721.913,E2 -3721.913} C_VEL
LIN {X 0,Y 545.169,Z 292.524,A -85,B 0,C 180,E1 -3724.556,E2 -3724.556} C_VEL
LIN {X 0,Y 545.268,Z 287.196,A -85,B 0,C 180,E1 -3727.284,E2 -3727.284} C_VEL
LIN {X 0,Y 545.41,Z 281.14,A -85,B 0,C 180,E1 -3730.513,E2 -3730.513} C_VEL
LIN {X 0,Y 545.1,Z 277.213,A -85,B 0,C 180,E1 -3732.782,E2 -3732.782} C_VEL
LIN {X 0,Y 545.046,Z 277.22,A -85,B 0,C 180,E1 -3735.87,E2 -3735.87} C_VEL
LIN {X 0,Y 545.084,Z 277.215,A -85,B 0,C 180,E1 -3738.886,E2 -3738.886} C_VEL
LIN {X 0,Y 545.049,Z 277.221,A -85,B 0,C 180,E1 -3741.762,E2 -3741.762} C_VEL
LIN {X 0,Y 545.019,Z 277.222,A -85,B 0,C 180,E1 -3744.53,E2 -3744.53} C_VEL
LIN {X 0,Y 545.073,Z 277.214,A -85,B 0,C 180,E1 -3747.212,E2 -3747.212} C_VEL
LIN {X 0,Y 545.058,Z 277.216,A -85,B 0,C 180,E1 -3749.81,E2 -3749.81} C_VEL
LIN {X 0,Y 545.075,Z 277.214,A -85,B 0,C 180,E1 -3752.828,E2 -3752.828} C_VEL
LIN {X 0,Y 545.045,Z 277.22,A -85,B 0,C 180,E1 -3755.631,E2 -3755.631} C_VEL
LIN {X 0,Y 545.056,Z 277.217,A -85,B 0,C 180,E1 -3758.836,E2 -3758.836} C_VEL
LIN {X 0,Y 545.076,Z 277.213,A -85,B 0,C 180,E1 -3761.196,E2 -3761.196} C_VEL
LIN {X 0,Y 545.064,Z 277.215,A -85,B 0,C 180,E1 -3763.521,E2 -3763.521} C_VEL
LIN {X 0,Y 545.079,Z 277.212,A -85,B 0,C 180,E1 -3765.82,E2 -3765.82} C_VEL
LIN {X 0,Y 545.125,Z 277.206,A -85,B 0,C 180,E1 -3768.85,E2 -3768.85} C_VEL
LIN {X 0,Y 545.117,Z 277.207,A -85,B 0,C 180,E1 -3771.847,E2 -3771.847} C_VEL
LIN {X 0,Y 545.198,Z 277.196,A -85,B 0,C 180,E1 -3774.823,E2 -3774.823} C_VEL
LIN {X 0,Y 545.192,Z 277.196,A -85,B 0,C 180,E1 -3777.784,E2 -3777.784} C_VEL
LIN {X 0,Y 545.196,Z 277.197,A -85,B 0,C 180,E1 -3780.739,E2 -3780.739} C_VEL
LIN {X 0,Y 545.166,Z 277.205,A -85,B 0,C 180,E1 -3782.956,E2 -3782.956} C_VEL
LIN {X 0,Y 545.154,Z 277.205,A -85,B 0,C 180,E1 -3785.92,E2 -3785.92} C_VEL
LIN {X 0,Y 545.11,Z 277.209,A -85,B 0,C 180,E1 -3788.9,E2 -3788.9} C_VEL
LIN {X 0,Y 545.126,Z 277.206,A -85,B 0,C 180,E1 -3791.904,E2 -3791.904} C_VEL
LIN {X 0,Y 545.073,Z 277.213,A -85,B 0,C 180,E1 -3794.944,E2 -3794.944} C_VEL
LIN {X 0,Y 545.075,Z 277.213,A -85,B 0,C 180,E1 -3798.026,E2 -3798.026} C_VEL
LIN {X 0,Y 545.085,Z 277.211,A -85,B 0,C 180,E1 -3800.373,E2 -3800.373} C_VEL
LIN {X 0,Y 545.084,Z 277.211,A -85,B 0,C 180,E1 -3803.559,E2 -3803.559} C_VEL
LIN {X 0,Y 545.072,Z 277.217,A -85,B 0,C 180,E1 -3806.001,E2 -3806.001} C_VEL
LIN {X 0,Y 545.067,Z 277.214,A -85,B 0,C 180,E1 -3808.746,E2 -3808.746} C_VEL
LIN {X 0,Y 545.071,Z 277.212,A -85,B 0,C 180,E1 -3811.683,E2 -3811.683} C_VEL
LIN {X 0,Y 545.051,Z 277.214,A -85,B 0,C 180,E1 -3814.565,E2 -3814.565} C_VEL
LIN {X 0,Y 545.055,Z 277.217,A -85,B 0,C 180,E1 -3816.99,E2 -3816.99} C_VEL
LIN {X 0,Y 544.35,Z 277.303,A -85,B 0,C 180,E1 -3817.606,E2 -3817.606} C_VEL
LIN {X 0,Y 541.489,Z 277.661,A -85,B 0,C 180,E1 -3818.607,E2 -3818.607} C_VEL
LIN {X 0,Y 539.102,Z 277.959,A -85,B 0,C 180,E1 -3819.413,E2 -3819.413} C_VEL
LIN {X 0,Y 538.091,Z 278.085,A -85,B 0,C 180,E1 -3820.035,E2 -3820.035} C_VEL
LIN {X 0,Y 538.015,Z 278.092,A -85,B 0,C 180,E1 -3820.246,E2 -3820.246} C_VEL
LIN {X 0,Y 538.021,Z 278.094,A -85,B 0,C 180,E1 -3822.988,E2 -3822.988} C_VEL
LIN {X 0,Y 538.025,Z 278.095,A -85,B 0,C 180,E1 -3825.926,E2 -3825.926} C_VEL
LIN {X 0,Y 537.999,Z 278.098,A -85,B 0,C 180,E1 -3827.213,E2 -3827.213} C_VEL
LIN {X 0,Y 538.048,Z 278.683,A -85,B 0,C 180,E1 -3828.23,E2 -3828.23} C_VEL
LIN {X 0,Y 538.117,Z 281.979,A -85,B 0,C 180,E1 -3830.404,E2 -3830.404} C_VEL
LIN {X 0,Y 538.081,Z 286.144,A -85,B 0,C 180,E1 -3833.073,E2 -3833.073} C_VEL
LIN {X 0,Y 537.996,Z 290.603,A -85,B 0,C 180,E1 -3835.826,E2 -3835.826} C_VEL
LIN {X 0,Y 537.904,Z 295.048,A -85,B 0,C 180,E1 -3838.493,E2 -3838.493} C_VEL
LIN {X 0,Y 537.869,Z 299.503,A -85,B 0,C 180,E1 -3841.098,E2 -3841.098} C_VEL
LIN {X 0,Y 537.768,Z 305.405,A -85,B 0,C 180,E1 -3844.452,E2 -3844.452} C_VEL
LIN {X 0,Y 537.659,Z 309.822,A -85,B 0,C 180,E1 -3846.913,E2 -3846.913} C_VEL
LIN {X 0,Y 537.588,Z 314.243,A -85,B 0,C 180,E1 -3849.331,E2 -3849.331} C_VEL
LIN {X 0,Y 537.606,Z 317.771,A -85,B 0,C 180,E1 -3851.235,E2 -3851.235} C_VEL
LIN {X 0,Y 540.908,Z 331.186,A -85,B 0,C 180,E1 -3851.606,E2 -3851.606} C_VEL
LIN {X 0,Y 540.674,Z 345.839,A -85,B 0,C 180,E1 -3851.999,E2 -3851.999} C_VEL
LIN {X 0,Y 540.329,Z 360.049,A -85,B 0,C 180,E1 -3852.524,E2 -3852.524} C_VEL
LIN {X 0,Y 539.967,Z 373.546,A -85,B 0,C 180,E1 -3853.167,E2 -3853.167} C_VEL
LIN {X 0,Y 539.609,Z 386.54,A -85,B 0,C 180,E1 -3853.933,E2 -3853.933} C_VEL
LIN {X 0,Y 539.208,Z 399.816,A -85,B 0,C 180,E1 -3854.89,E2 -3854.89} C_VEL
LIN {X 0,Y 538.868,Z 410.922,A -85,B 0,C 180,E1 -3855.846,E2 -3855.846} C_VEL
LIN {X 0,Y 538.547,Z 422.112,A -85,B 0,C 180,E1 -3856.991,E2 -3856.991} C_VEL
LIN {X 0,Y 538.184,Z 433.201,A -85,B 0,C 180,E1 -3858.352,E2 -3858.352} C_VEL
LIN {X 0,Y 538.018,Z 442.02,A -85,B 0,C 180,E1 -3859.653,E2 -3859.653} C_VEL
LIN {X 0,Y 537.799,Z 449.507,A -85,B 0,C 180,E1 -3860.978,E2 -3860.978} C_VEL
LIN {X 0,Y 537.662,Z 456.51,A -85,B 0,C 180,E1 -3862.49,E2 -3862.49} C_VEL
LIN {X 0,Y 537.62,Z 462.018,A -85,B 0,C 180,E1 -3863.997,E2 -3863.997} C_VEL
LIN {X 0,Y 537.507,Z 466.183,A -85,B 0,C 180,E1 -3865.501,E2 -3865.501} C_VEL
LIN {X 0,Y 537.543,Z 469.114,A -85,B 0,C 180,E1 -3867.003,E2 -3867.003} C_VEL
LIN {X 0,Y 537.448,Z 470.879,A -85,B 0,C 180,E1 -3868.502,E2 -3868.502} C_VEL
LIN {X 0,Y 537.44,Z 471.496,A -85,B 0,C 180,E1 -3870,E2 -3870} C_VEL
LIN {X 0,Y 537.449,Z 470.938,A -85,B 0,C 180,E1 -3871.499,E2 -3871.499} C_VEL
LIN {X 0,Y 537.545,Z 469.252,A -85,B 0,C 180,E1 -3872.998,E2 -3872.998} C_VEL
LIN {X 0,Y 537.507,Z 466.398,A -85,B 0,C 180,E1 -3874.5,E2 -3874.5} C_VEL
LIN {X 0,Y 537.594,Z 462.31,A -85,B 0,C 180,E1 -3876.003,E2 -3876.003} C_VEL
LIN {X 0,Y 537.662,Z 456.891,A -85,B 0,C 180,E1 -3877.511,E2 -3877.511} C_VEL
LIN {X 0,Y 537.797,Z 449.988,A -85,B 0,C 180,E1 -3879.022,E2 -3879.022} C_VEL
LIN {X 0,Y 538.022,Z 441.375,A -85,B 0,C 180,E1 -3880.538,E2 -3880.538} C_VEL
LIN {X 0,Y 538.217,Z 431.901,A -85,B 0,C 180,E1 -3881.91,E2 -3881.91} C_VEL
LIN {X 0,Y 538.54,Z 421.165,A -85,B 0,C 180,E1 -3883.202,E2 -3883.202} C_VEL
LIN {X 0,Y 538.908,Z 409.787,A -85,B 0,C 180,E1 -3884.346,E2 -3884.346} C_VEL
LIN {X 0,Y 539.292,Z 397.359,A -85,B 0,C 180,E1 -3885.391,E2 -3885.391} C_VEL
LIN {X 0,Y 539.688,Z 384.978,A -85,B 0,C 180,E1 -3886.259,E2 -3886.259} C_VEL
LIN {X 0,Y 540.042,Z 371.643,A -85,B 0,C 180,E1 -3887.026,E2 -3887.026} C_VEL
LIN {X 0,Y 540.431,Z 358.269,A -85,B 0,C 180,E1 -3887.639,E2 -3887.639} C_VEL
LIN {X 0,Y 540.702,Z 343.823,A -85,B 0,C 180,E1 -3888.154,E2 -3888.154} C_VEL
LIN {X 0,Y 540.819,Z 330.736,A -85,B 0,C 180,E1 -3888.497,E2 -3888.497} C_VEL
LIN {X 0,Y 537.611,Z 317.75,A -85,B 0,C 180,E1 -3888.865,E2 -3888.865} C_VEL
LIN {X 0,Y 537.647,Z 312.216,A -85,B 0,C 180,E1 -3891.86,E2 -3891.86} C_VEL
LIN {X 0,Y 537.755,Z 307.04,A -85,B 0,C 180,E1 -3894.722,E2 -3894.722} C_VEL
LIN {X 0,Y 537.819,Z 301.16,A -85,B 0,C 180,E1 -3898.062,E2 -3898.062} C_VEL
LIN {X 0,Y 537.892,Z 296.696,A -85,B 0,C 180,E1 -3900.635,E2 -3900.635} C_VEL
LIN {X 0,Y 537.997,Z 292.236,A -85,B 0,C 180,E1 -3903.275,E2 -3903.275} C_VEL
LIN {X 0,Y 538.046,Z 287.778,A -85,B 0,C 180,E1 -3906,E2 -3906} C_VEL
LIN {X 0,Y 538.105,Z 283.304,A -85,B 0,C 180,E1 -3908.822,E2 -3908.822} C_VEL
LIN {X 0,Y 538.136,Z 280.324,A -85,B 0,C 180,E1 -3910.767,E2 -3910.767} C_VEL
LIN {X 0,Y 538.04,Z 278.664,A -85,B 0,C 180,E1 -3911.88,E2 -3911.88} C_VEL
LIN {X 0,Y 537.997,Z 278.098,A -85,B 0,C 180,E1 -3912.984,E2 -3912.984} C_VEL
LIN {X 0,Y 538.02,Z 278.096,A -85,B 0,C 180,E1 -3915.926,E2 -3915.926} C_VEL
LIN {X 0,Y 538.046,Z 278.088,A -85,B 0,C 180,E1 -3919.224,E2 -3919.224} C_VEL
LIN {X 0,Y 537.992,Z 278.097,A -85,B 0,C 180,E1 -3922.122,E2 -3922.122} C_VEL
LIN {X 0,Y 537.989,Z 278.1,A -85,B 0,C 180,E1 -3924.915,E2 -3924.915} C_VEL
LIN {X 0,Y 538.017,Z 278.094,A -85,B 0,C 180,E1 -3927.617,E2 -3927.617} C_VEL
LIN {X 0,Y 538.012,Z 278.092,A -85,B 0,C 180,E1 -3930.238,E2 -3930.238} C_VEL
LIN {X 0,Y 538.027,Z 278.092,A -85,B 0,C 180,E1 -3932.794,E2 -3932.794} C_VEL
LIN {X 0,Y 538.022,Z 278.093,A -85,B 0,C 180,E1 -3935.291,E2 -3935.291} C_VEL
LIN {X 0,Y 538.012,Z 278.091,A -85,B 0,C 180,E1 -3938.042,E2 -3938.042} C_VEL
LIN {X 0,Y 538.031,Z 278.088,A -85,B 0,C 180,E1 -3940.94,E2 -3940.94} C_VEL
LIN {X 0,Y 538.021,Z 278.094,A -85,B 0,C 180,E1 -3943.299,E2 -3943.299} C_VEL
LIN {X 0,Y 538.05,Z 278.087,A -85,B 0,C 180,E1 -3945.63,E2 -3945.63} C_VEL
LIN {X 0,Y 538.074,Z 278.084,A -85,B 0,C 180,E1 -3948.701,E2 -3948.701} C_VEL
LIN {X 0,Y 538.08,Z 278.083,A -85,B 0,C 180,E1 -3951.739,E2 -3951.739} C_VEL
LIN {X 0,Y 538.156,Z 278.074,A -85,B 0,C 180,E1 -3954.755,E2 -3954.755} C_VEL
LIN {X 0,Y 538.167,Z 278.072,A -85,B 0,C 180,E1 -3957.755,E2 -3957.755} C_VEL
LIN {X 0,Y 538.17,Z 278.072,A -85,B 0,C 180,E1 -3960.748,E2 -3960.748} C_VEL
LIN {X 0,Y 538.136,Z 278.081,A -85,B 0,C 180,E1 -3962.994,E2 -3962.994} C_VEL
LIN {X 0,Y 538.108,Z 278.083,A -85,B 0,C 180,E1 -3965.997,E2 -3965.997} C_VEL
LIN {X 0,Y 538.065,Z 278.088,A -85,B 0,C 180,E1 -3969.018,E2 -3969.018} C_VEL
LIN {X 0,Y 538.078,Z 278.087,A -85,B 0,C 180,E1 -3972.063,E2 -3972.063} C_VEL
LIN {X 0,Y 538.038,Z 278.092,A -85,B 0,C 180,E1 -3975.144,E2 -3975.144} C_VEL
LIN {X 0,Y 538.029,Z 278.094,A -85,B 0,C 180,E1 -3978.27,E2 -3978.27} C_VEL
LIN {X 0,Y 538.032,Z 278.089,A -85,B 0,C 180,E1 -3980.652,E2 -3980.652} C_VEL
LIN {X 0,Y 538,Z 278.093,A -85,B 0,C 180,E1 -3983.888,E2 -3983.888} C_VEL
LIN {X 0,Y 538.035,Z 278.091,A -85,B 0,C 180,E1 -3986.367,E2 -3986.367} C_VEL
LIN {X 0,Y 538.026,Z 278.095,A -85,B 0,C 180,E1 -3988.933,E2 -3988.933} C_VEL
LIN {X 0,Y 538.008,Z 278.096,A -85,B 0,C 180,E1 -3991.888,E2 -3991.888} C_VEL
LIN {X 0,Y 538.004,Z 278.095,A -85,B 0,C 180,E1 -3994.617,E2 -3994.617} C_VEL
LIN {X 0,Y 538,Z 278.096,A -85,B 0,C 180,E1 -3997.17,E2 -3997.17} C_VEL
LIN {X 0,Y 538.024,Z 278.096,A -85,B 0,C 180,E1 -3999.797,E2 -3999.797} C_VEL
LIN {X 0,Y 537.997,Z 278.099,A -85,B 0,C 180,E1 -4002.788,E2 -4002.788} C_VEL
LIN {X 0,Y 538.03,Z 278.095,A -85,B 0,C 180,E1 -4005.141,E2 -4005.141} C_VEL
LIN {X 0,Y 538.078,Z 278.202,A -85,B 0,C 180,E1 -4007.146,E2 -4007.146} C_VEL
LIN {X 0,Y 538.41,Z 281.86,A -85,B 0,C 180,E1 -4009.258,E2 -4009.258} C_VEL
LIN {X 0,Y 538.274,Z 287.162,A -85,B 0,C 180,E1 -4012.146,E2 -4012.146} C_VEL
LIN {X 0,Y 538.163,Z 292.489,A -85,B 0,C 180,E1 -4014.928,E2 -4014.928} C_VEL
LIN {X 0,Y 538.051,Z 297.823,A -85,B 0,C 180,E1 -4017.62,E2 -4017.62} C_VEL
LIN {X 0,Y 537.971,Z 303.174,A -85,B 0,C 180,E1 -4020.236,E2 -4020.236} C_VEL
LIN {X 0,Y 537.872,Z 308.561,A -85,B 0,C 180,E1 -4022.786,E2 -4022.786} C_VEL
LIN {X 0,Y 537.797,Z 313.936,A -85,B 0,C 180,E1 -4025.28,E2 -4025.28} C_VEL
LIN {X 0,Y 537.753,Z 321.08,A -85,B 0,C 180,E1 -4028.535,E2 -4028.535} C_VEL
LIN {X 0,Y 537.672,Z 327.029,A -85,B 0,C 180,E1 -4031.191,E2 -4031.191} C_VEL
LIN {X 0,Y 540.918,Z 341.037,A -85,B 0,C 180,E1 -4031.559,E2 -4031.559} C_VEL
LIN {X 0,Y 540.653,Z 356.065,A -85,B 0,C 180,E1 -4031.961,E2 -4031.961} C_VEL
LIN {X 0,Y 540.298,Z 370.932,A -85,B 0,C 180,E1 -4032.516,E2 -4032.516} C_VEL
LIN {X 0,Y 539.947,Z 384.359,A -85,B 0,C 180,E1 -4033.165,E2 -4033.165} C_VEL
LIN {X 0,Y 539.533,Z 398.617,A -85,B 0,C 180,E1 -4034.027,E2 -4034.027} C_VEL
LIN {X 0,Y 539.162,Z 411.52,A -85,B 0,C 180,E1 -4034.985,E2 -4034.985} C_VEL
LIN {X 0,Y 538.755,Z 423.326,A -85,B 0,C 180,E1 -4036.035,E2 -4036.035} C_VEL
LIN {X 0,Y 538.462,Z 434.137,A -85,B 0,C 180,E1 -4037.18,E2 -4037.18} C_VEL
LIN {X 0,Y 538.13,Z 443.72,A -85,B 0,C 180,E1 -4038.379,E2 -4038.379} C_VEL
LIN {X 0,Y 538.017,Z 452.295,A -85,B 0,C 180,E1 -4039.653,E2 -4039.653} C_VEL
LIN {X 0,Y 537.797,Z 459.749,A -85,B 0,C 180,E1 -4040.978,E2 -4040.978} C_VEL
LIN {X 0,Y 537.661,Z 466.7,A -85,B 0,C 180,E1 -4042.489,E2 -4042.489} C_VEL
LIN {X 0,Y 537.623,Z 472.162,A -85,B 0,C 180,E1 -4043.997,E2 -4043.997} C_VEL
LIN {X 0,Y 537.508,Z 476.291,A -85,B 0,C 180,E1 -4045.5,E2 -4045.5} C_VEL
LIN {X 0,Y 537.543,Z 479.184,A -85,B 0,C 180,E1 -4047.002,E2 -4047.002} C_VEL
LIN {X 0,Y 537.448,Z 480.909,A -85,B 0,C 180,E1 -4048.501,E2 -4048.501} C_VEL
LIN {X 0,Y 537.439,Z 481.5,A -85,B 0,C 180,E1 -4050,E2 -4050} C_VEL
LIN {X 0,Y 537.448,Z 480.908,A -85,B 0,C 180,E1 -4051.498,E2 -4051.498} C_VEL
LIN {X 0,Y 537.543,Z 479.181,A -85,B 0,C 180,E1 -4052.997,E2 -4052.997} C_VEL
LIN {X 0,Y 537.508,Z 476.29,A -85,B 0,C 180,E1 -4054.499,E2 -4054.499} C_VEL
LIN {X 0,Y 537.623,Z 472.167,A -85,B 0,C 180,E1 -4056.003,E2 -4056.003} C_VEL
LIN {X 0,Y 537.66,Z 466.703,A -85,B 0,C 180,E1 -4057.51,E2 -4057.51} C_VEL
LIN {X 0,Y 537.797,Z 459.747,A -85,B 0,C 180,E1 -4059.022,E2 -4059.022} C_VEL
LIN {X 0,Y 538.023,Z 451.085,A -85,B 0,C 180,E1 -4060.537,E2 -4060.537} C_VEL
LIN {X 0,Y 538.228,Z 441.537,A -85,B 0,C 180,E1 -4061.911,E2 -4061.911} C_VEL
LIN {X 0,Y 538.524,Z 432.512,A -85,B 0,C 180,E1 -4063.009,E2 -4063.009} C_VEL
LIN {X 0,Y 538.871,Z 420.365,A -85,B 0,C 180,E1 -4064.25,E2 -4064.25} C_VEL
LIN {X 0,Y 539.282,Z 408.507,A -85,B 0,C 180,E1 -4065.26,E2 -4065.26} C_VEL
LIN {X 0,Y 539.632,Z 395.775,A -85,B 0,C 180,E1 -4066.163,E2 -4066.163} C_VEL
LIN {X 0,Y 540.013,Z 382.597,A -85,B 0,C 180,E1 -4066.929,E2 -4066.929} C_VEL
LIN {X 0,Y 540.401,Z 369.199,A -85,B 0,C 180,E1 -4067.555,E2 -4067.555} C_VEL
LIN {X 0,Y 540.671,Z 354.476,A -85,B 0,C 180,E1 -4068.09,E2 -4068.09} C_VEL
LIN {X 0,Y 540.886,Z 340.037,A -85,B 0,C 180,E1 -4068.464,E2 -4068.464} C_VEL
LIN {X 0,Y 537.659,Z 326.977,A -85,B 0,C 180,E1 -4068.829,E2 -4068.829} C_VEL
LIN {X 0,Y 537.743,Z 321.062,A -85,B 0,C 180,E1 -4071.465,E2 -4071.465} C_VEL
LIN {X 0,Y 537.795,Z 313.901,A -85,B 0,C 180,E1 -4074.719,E2 -4074.719} C_VEL
LIN {X 0,Y 537.867,Z 308.317,A -85,B 0,C 180,E1 -4077.313,E2 -4077.313} C_VEL
LIN {X 0,Y 537.968,Z 303.18,A -85,B 0,C 180,E1 -4079.763,E2 -4079.763} C_VEL
LIN {X 0,Y 538.049,Z 297.827,A -85,B 0,C 180,E1 -4082.38,E2 -4082.38} C_VEL
LIN {X 0,Y 538.161,Z 292.491,A -85,B 0,C 180,E1 -4085.071,E2 -4085.071} C_VEL
LIN {X 0,Y 538.277,Z 287.169,A -85,B 0,C 180,E1 -4087.853,E2 -4087.853} C_VEL
LIN {X 0,Y 538.401,Z 281.767,A -85,B 0,C 180,E1 -4090.791,E2 -4090.791} C_VEL
LIN {X 0,Y 538.058,Z 278.09,A -85,B 0,C 180,E1 -4092.991,E2 -4092.991} C_VEL
LIN {X 0,Y 538.015,Z 278.095,A -85,B 0,C 180,E1 -4095.926,E2 -4095.926} C_VEL
LIN {X 0,Y 538.044,Z 278.089,A -85,B 0,C 180,E1 -4099.224,E2 -4099.224} C_VEL
LIN {X 0,Y 537.987,Z 278.097,A -85,B 0,C 180,E1 -4102.122,E2 -4102.122} C_VEL
LIN {X 0,Y 537.984,Z 278.101,A -85,B 0,C 180,E1 -4104.915,E2 -4104.915} C_VEL
LIN {X 0,Y 538.023,Z 278.095,A -85,B 0,C 180,E1 -4107.618,E2 -4107.618} C_VEL
LIN {X 0,Y 538.008,Z 278.094,A -85,B 0,C 180,E1 -4110.238,E2 -4110.238} C_VEL
LIN {X 0,Y 538.044,Z 278.09,A -85,B 0,C 180,E1 -4112.795,E2 -4112.795} C_VEL
LIN {X 0,Y 538.041,Z 278.091,A -85,B 0,C 180,E1 -4115.292,E2 -4115.292} C_VEL
LIN {X 0,Y 538.007,Z 278.093,A -85,B 0,C 180,E1 -4118.042,E2 -4118.042} C_VEL
LIN {X 0,Y 538.031,Z 278.089,A -85,B 0,C 180,E1 -4120.94,E2 -4120.94} C_VEL
LIN {X 0,Y 538.016,Z 278.095,A -85,B 0,C 180,E1 -4123.299,E2 -4123.299} C_VEL
LIN {X 0,Y 538.05,Z 278.086,A -85,B 0,C 180,E1 -4125.63,E2 -4125.63} C_VEL
LIN {X 0,Y 538.082,Z 278.083,A -85,B 0,C 180,E1 -4128.702,E2 -4128.702} C_VEL
LIN {X 0,Y 538.075,Z 278.083,A -85,B 0,C 180,E1 -4131.74,E2 -4131.74} C_VEL
LIN {X 0,Y 538.154,Z 278.073,A -85,B 0,C 180,E1 -4134.755,E2 -4134.755} C_VEL
LIN {X 0,Y 538.163,Z 278.071,A -85,B 0,C 180,E1 -4137.755,E2 -4137.755} C_VEL
LIN {X 0,Y 538.167,Z 278.072,A -85,B 0,C 180,E1 -4140.748,E2 -4140.748} C_VEL
LIN {X 0,Y 538.133,Z 278.081,A -85,B 0,C 180,E1 -4142.995,E2 -4142.995} C_VEL
LIN {X 0,Y 538.105,Z 278.084,A -85,B 0,C 180,E1 -4145.998,E2 -4145.998} C_VEL
LIN {X 0,Y 538.062,Z 278.088,A -85,B 0,C 180,E1 -4149.018,E2 -4149.018} C_VEL
LIN {X 0,Y 538.074,Z 278.086,A -85,B 0,C 180,E1 -4152.063,E2 -4152.063} C_VEL
LIN {X 0,Y 538.034,Z 278.092,A -85,B 0,C 180,E1 -4155.144,E2 -4155.144} C_VEL
LIN {X 0,Y 538.027,Z 278.093,A -85,B 0,C 180,E1 -4158.27,E2 -4158.27} C_VEL
LIN {X 0,Y 538.029,Z 278.089,A -85,B 0,C 180,E1 -4160.652,E2 -4160.652} C_VEL
LIN {X 0,Y 538.017,Z 278.091,A -85,B 0,C 180,E1 -4163.888,E2 -4163.888} C_VEL
LIN {X 0,Y 538.034,Z 278.09,A -85,B 0,C 180,E1 -4166.367,E2 -4166.367} C_VEL
LIN {X 0,Y 538.022,Z 278.094,A -85,B 0,C 180,E1 -4168.934,E2 -4168.934} C_VEL
LIN {X 0,Y 538.021,Z 278.092,A -85,B 0,C 180,E1 -4171.891,E2 -4171.891} C_VEL
LIN {X 0,Y 538.001,Z 278.092,A -85,B 0,C 180,E1 -4174.618,E2 -4174.618} C_VEL
LIN {X 0,Y 537.997,Z 278.094,A -85,B 0,C 180,E1 -4177.17,E2 -4177.17} C_VEL
LIN {X 0,Y 538.015,Z 278.092,A -85,B 0,C 180,E1 -4180.246,E2 -4180.246} C_VEL
LIN {X 0,Y 537.362,Z 278.175,A -85,B 0,C 180,E1 -4180.871,E2 -4180.871} C_VEL
LIN {X 0,Y 534.508,Z 278.529,A -85,B 0,C 180,E1 -4181.886,E2 -4181.886} C_VEL
LIN {X 0,Y 532.082,Z 278.835,A -85,B 0,C 180,E1 -4182.703,E2 -4182.703} C_VEL
LIN {X 0,Y 531.035,Z 278.962,A -85,B 0,C 180,E1 -4183.334,E2 -4183.334} C_VEL
LIN {X 0,Y 530.948,Z 278.972,A -85,B 0,C 180,E1 -4183.548,E2 -4183.548} C_VEL
LIN {X 0,Y 530.951,Z 278.974,A -85,B 0,C 180,E1 -4186.505,E2 -4186.505} C_VEL
LIN {X 0,Y 530.949,Z 279.147,A -85,B 0,C 180,E1 -4187.838,E2 -4187.838} C_VEL
LIN {X 0,Y 531.098,Z 282.539,A -85,B 0,C 180,E1 -4190.131,E2 -4190.131} C_VEL
LIN {X 0,Y 531.055,Z 286.285,A -85,B 0,C 180,E1 -4192.565,E2 -4192.565} C_VEL
LIN {X 0,Y 530.987,Z 290.641,A -85,B 0,C 180,E1 -4195.311,E2 -4195.311} C_VEL
LIN {X 0,Y 530.878,Z 295.088,A -85,B 0,C 180,E1 -4198.027,E2 -4198.027} C_VEL
LIN {X 0,Y 530.798,Z 299.942,A -85,B 0,C 180,E1 -4200.912,E2 -4200.912} C_VEL
LIN {X 0,Y 530.683,Z 303.967,A -85,B 0,C 180,E1 -4203.24,E2 -4203.24} C_VEL
LIN {X 0,Y 530.667,Z 308.893,A -85,B 0,C 180,E1 -4206.038,E2 -4206.038} C_VEL
LIN {X 0,Y 530.539,Z 314.301,A -85,B 0,C 180,E1 -4209.044,E2 -4209.044} C_VEL
LIN {X 0,Y 530.54,Z 317.829,A -85,B 0,C 180,E1 -4210.972,E2 -4210.972} C_VEL
LIN {X 0,Y 534.143,Z 332.823,A -85,B 0,C 180,E1 -4211.398,E2 -4211.398} C_VEL
LIN {X 0,Y 533.891,Z 348.036,A -85,B 0,C 180,E1 -4211.831,E2 -4211.831} C_VEL
LIN {X 0,Y 533.5,Z 362.857,A -85,B 0,C 180,E1 -4212.413,E2 -4212.413} C_VEL
LIN {X 0,Y 533.09,Z 377.132,A -85,B 0,C 180,E1 -4213.14,E2 -4213.14} C_VEL
LIN {X 0,Y 532.678,Z 389.429,A -85,B 0,C 180,E1 -4213.915,E2 -4213.915} C_VEL
LIN {X 0,Y 532.234,Z 402.178,A -85,B 0,C 180,E1 -4214.883,E2 -4214.883} C_VEL
LIN {X 0,Y 531.845,Z 412.884,A -85,B 0,C 180,E1 -4215.85,E2 -4215.85} C_VEL
LIN {X 0,Y 531.51,Z 423.765,A -85,B 0,C 180,E1 -4217.01,E2 -4217.01} C_VEL
LIN {X 0,Y 531.14,Z 433.82,A -85,B 0,C 180,E1 -4218.283,E2 -4218.283} C_VEL
LIN {X 0,Y 530.942,Z 443.154,A -85,B 0,C 180,E1 -4219.707,E2 -4219.707} C_VEL
LIN {X 0,Y 530.765,Z 449.51,A -85,B 0,C 180,E1 -4220.858,E2 -4220.858} C_VEL
LIN {X 0,Y 530.602,Z 456.513,A -85,B 0,C 180,E1 -4222.389,E2 -4222.389} C_VEL
LIN {X 0,Y 530.526,Z 462.02,A -85,B 0,C 180,E1 -4223.917,E2 -4223.917} C_VEL
LIN {X 0,Y 530.412,Z 466.184,A -85,B 0,C 180,E1 -4225.441,E2 -4225.441} C_VEL
LIN {X 0,Y 530.448,Z 469.114,A -85,B 0,C 180,E1 -4226.962,E2 -4226.962} C_VEL
LIN {X 0,Y 530.358,Z 470.879,A -85,B 0,C 180,E1 -4228.482,E2 -4228.482} C_VEL
LIN {X 0,Y 530.341,Z 471.497,A -85,B 0,C 180,E1 -4230,E2 -4230} C_VEL
LIN {X 0,Y 530.359,Z 470.937,A -85,B 0,C 180,E1 -4231.519,E2 -4231.519} C_VEL
LIN {X 0,Y 530.45,Z 469.25,A -85,B 0,C 180,E1 -4233.038,E2 -4233.038} C_VEL
LIN {X 0,Y 530.412,Z 466.396,A -85,B 0,C 180,E1 -4234.56,E2 -4234.56} C_VEL
LIN {X 0,Y 530.502,Z 462.308,A -85,B 0,C 180,E1 -4236.084,E2 -4236.084} C_VEL
LIN {X 0,Y 530.602,Z 456.888,A -85,B 0,C 180,E1 -4237.612,E2 -4237.612} C_VEL
LIN {X 0,Y 530.76,Z 449.984,A -85,B 0,C 180,E1 -4239.143,E2 -4239.143} C_VEL
LIN {X 0,Y 530.98,Z 442.558,A -85,B 0,C 180,E1 -4240.486,E2 -4240.486} C_VEL
LIN {X 0,Y 531.192,Z 433.568,A -85,B 0,C 180,E1 -4241.842,E2 -4241.842} C_VEL
LIN {X 0,Y 531.463,Z 424.514,A -85,B 0,C 180,E1 -4242.992,E2 -4242.992} C_VEL
LIN {X 0,Y 531.818,Z 413.774,A -85,B 0,C 180,E1 -4244.151,E2 -4244.151} C_VEL
LIN {X 0,Y 532.234,Z 402.066,A -85,B 0,C 180,E1 -4245.215,E2 -4245.215} C_VEL
LIN {X 0,Y 532.665,Z 389.296,A -85,B 0,C 180,E1 -4246.184,E2 -4246.184} C_VEL
LIN {X 0,Y 533.128,Z 375.211,A -85,B 0,C 180,E1 -4247.056,E2 -4247.056} C_VEL
LIN {X 0,Y 533.547,Z 362.032,A -85,B 0,C 180,E1 -4247.712,E2 -4247.712} C_VEL
LIN {X 0,Y 533.898,Z 346.975,A -85,B 0,C 180,E1 -4248.293,E2 -4248.293} C_VEL
LIN {X 0,Y 534.09,Z 331.935,A -85,B 0,C 180,E1 -4248.713,E2 -4248.713} C_VEL
LIN {X 0,Y 530.545,Z 317.845,A -85,B 0,C 180,E1 -4249.113,E2 -4249.113} C_VEL
LIN {X 0,Y 530.573,Z 312.6,A -85,B 0,C 180,E1 -4251.994,E2 -4251.994} C_VEL
LIN {X 0,Y 530.666,Z 308.584,A -85,B 0,C 180,E1 -4254.24,E2 -4254.24} C_VEL
LIN {X 0,Y 530.682,Z 304.174,A -85,B 0,C 180,E1 -4256.761,E2 -4256.761} C_VEL
LIN {X 0,Y 530.793,Z 299.708,A -85,B 0,C 180,E1 -4259.334,E2 -4259.334} C_VEL
LIN {X 0,Y 530.88,Z 295.065,A -85,B 0,C 180,E1 -4262.085,E2 -4262.085} C_VEL
LIN {X 0,Y 530.98,Z 290.525,A -85,B 0,C 180,E1 -4264.852,E2 -4264.852} C_VEL
LIN {X 0,Y 531.057,Z 286.318,A -85,B 0,C 180,E1 -4267.5,E2 -4267.5} C_VEL
LIN {X 0,Y 531.098,Z 281.844,A -85,B 0,C 180,E1 -4270.422,E2 -4270.422} C_VEL
LIN {X 0,Y 530.94,Z 278.978,A -85,B 0,C 180,E1 -4272.46,E2 -4272.46} C_VEL
LIN {X 0,Y 530.985,Z 278.972,A -85,B 0,C 180,E1 -4275.453,E2 -4275.453} C_VEL
LIN {X 0,Y 530.991,Z 278.97,A -85,B 0,C 180,E1 -4278.564,E2 -4278.564} C_VEL
LIN {X 0,Y 530.959,Z 278.973,A -85,B 0,C 180,E1 -4281.529,E2 -4281.529} C_VEL
LIN {X 0,Y 530.946,Z 278.974,A -85,B 0,C 180,E1 -4284.379,E2 -4284.379} C_VEL
LIN {X 0,Y 530.965,Z 278.97,A -85,B 0,C 180,E1 -4287.133,E2 -4287.133} C_VEL
LIN {X 0,Y 530.966,Z 278.972,A -85,B 0,C 180,E1 -4289.803,E2 -4289.803} C_VEL
LIN {X 0,Y 530.969,Z 278.974,A -85,B 0,C 180,E1 -4292.476,E2 -4292.476} C_VEL
LIN {X 0,Y 530.986,Z 278.967,A -85,B 0,C 180,E1 -4294.941,E2 -4294.941} C_VEL
LIN {X 0,Y 530.974,Z 278.967,A -85,B 0,C 180,E1 -4297.898,E2 -4297.898} C_VEL
LIN {X 0,Y 530.99,Z 278.966,A -85,B 0,C 180,E1 -4300.677,E2 -4300.677} C_VEL
LIN {X 0,Y 530.982,Z 278.971,A -85,B 0,C 180,E1 -4303.071,E2 -4303.071} C_VEL
LIN {X 0,Y 531.008,Z 278.964,A -85,B 0,C 180,E1 -4305.435,E2 -4305.435} C_VEL
LIN {X 0,Y 531.032,Z 278.961,A -85,B 0,C 180,E1 -4308.55,E2 -4308.55} C_VEL
LIN {X 0,Y 531.05,Z 278.958,A -85,B 0,C 180,E1 -4311.629,E2 -4311.629} C_VEL
LIN {X 0,Y 531.114,Z 278.951,A -85,B 0,C 180,E1 -4314.685,E2 -4314.685} C_VEL
LIN {X 0,Y 531.138,Z 278.948,A -85,B 0,C 180,E1 -4317.725,E2 -4317.725} C_VEL
LIN {X 0,Y 531.141,Z 278.947,A -85,B 0,C 180,E1 -4320.758,E2 -4320.758} C_VEL
LIN {X 0,Y 531.103,Z 278.957,A -85,B 0,C 180,E1 -4323.034,E2 -4323.034} C_VEL
LIN {X 0,Y 531.062,Z 278.962,A -85,B 0,C 180,E1 -4326.077,E2 -4326.077} C_VEL
LIN {X 0,Y 531.026,Z 278.967,A -85,B 0,C 180,E1 -4329.138,E2 -4329.138} C_VEL
LIN {X 0,Y 531.035,Z 278.966,A -85,B 0,C 180,E1 -4332.225,E2 -4332.225} C_VEL
LIN {X 0,Y 530.989,Z 278.972,A -85,B 0,C 180,E1 -4335.35,E2 -4335.35} C_VEL
LIN {X 0,Y 530.987,Z 278.971,A -85,B 0,C 180,E1 -4338.521,E2 -4338.521} C_VEL
LIN {X 0,Y 530.993,Z 278.967,A -85,B 0,C 180,E1 -4340.938,E2 -4340.938} C_VEL
LIN {X 0,Y 530.968,Z 278.971,A -85,B 0,C 180,E1 -4344.225,E2 -4344.225} C_VEL
LIN {X 0,Y 530.993,Z 278.966,A -85,B 0,C 180,E1 -4346.744,E2 -4346.744} C_VEL
LIN {X 0,Y 530.975,Z 278.973,A -85,B 0,C 180,E1 -4349.323,E2 -4349.323} C_VEL
LIN {X 0,Y 530.963,Z 278.976,A -85,B 0,C 180,E1 -4352.101,E2 -4352.101} C_VEL
LIN {X 0,Y 530.962,Z 278.974,A -85,B 0,C 180,E1 -4354.85,E2 -4354.85} C_VEL
LIN {X 0,Y 530.963,Z 278.972,A -85,B 0,C 180,E1 -4357.508,E2 -4357.508} C_VEL
LIN {X 0,Y 530.979,Z 278.969,A -85,B 0,C 180,E1 -4360.433,E2 -4360.433} C_VEL
LIN {X 0,Y 530.943,Z 278.975,A -85,B 0,C 180,E1 -4363.497,E2 -4363.497} C_VEL
LIN {X 0,Y 530.974,Z 278.974,A -85,B 0,C 180,E1 -4366.507,E2 -4366.507} C_VEL
LIN {X 0,Y 531.021,Z 279.015,A -85,B 0,C 180,E1 -4366.928,E2 -4366.928} C_VEL
LIN {X 0,Y 531.371,Z 282.405,A -85,B 0,C 180,E1 -4368.928,E2 -4368.928} C_VEL
LIN {X 0,Y 531.293,Z 287.128,A -85,B 0,C 180,E1 -4371.558,E2 -4371.558} C_VEL
LIN {X 0,Y 531.168,Z 292.458,A -85,B 0,C 180,E1 -4374.397,E2 -4374.397} C_VEL
LIN {X 0,Y 531.043,Z 297.786,A -85,B 0,C 180,E1 -4377.139,E2 -4377.139} C_VEL
LIN {X 0,Y 530.923,Z 303.116,A -85,B 0,C 180,E1 -4379.8,E2 -4379.8} C_VEL
LIN {X 0,Y 530.821,Z 308.722,A -85,B 0,C 180,E1 -4382.507,E2 -4382.507} C_VEL
LIN {X 0,Y 530.72,Z 313.861,A -85,B 0,C 180,E1 -4384.928,E2 -4384.928} C_VEL
LIN {X 0,Y 530.67,Z 320.461,A -85,B 0,C 180,E1 -4387.98,E2 -4387.98} C_VEL
LIN {X 0,Y 530.619,Z 327.007,A -85,B 0,C 180,E1 -4390.933,E2 -4390.933} C_VEL
LIN {X 0,Y 534.14,Z 341.338,A -85,B 0,C 180,E1 -4391.324,E2 -4391.324} C_VEL
LIN {X 0,Y 533.881,Z 356.637,A -85,B 0,C 180,E1 -4391.745,E2 -4391.745} C_VEL
LIN {X 0,Y 533.506,Z 370.958,A -85,B 0,C 180,E1 -4392.29,E2 -4392.29} C_VEL
LIN {X 0,Y 533.14,Z 384.318,A -85,B 0,C 180,E1 -4392.944,E2 -4392.944} C_VEL
LIN {X 0,Y 532.674,Z 398.594,A -85,B 0,C 180,E1 -4393.816,E2 -4393.816} C_VEL
LIN {X 0,Y 532.256,Z 411.515,A -85,B 0,C 180,E1 -4394.785,E2 -4394.785} C_VEL
LIN {X 0,Y 531.819,Z 423.324,A -85,B 0,C 180,E1 -4395.849,E2 -4395.849} C_VEL
LIN {X 0,Y 531.493,Z 434.137,A -85,B 0,C 180,E1 -4397.009,E2 -4397.009} C_VEL
LIN {X 0,Y 531.107,Z 444.253,A -85,B 0,C 180,E1 -4398.299,E2 -4398.299} C_VEL
LIN {X 0,Y 530.941,Z 453.415,A -85,B 0,C 180,E1 -4399.706,E2 -4399.706} C_VEL
LIN {X 0,Y 530.76,Z 459.749,A -85,B 0,C 180,E1 -4400.857,E2 -4400.857} C_VEL
LIN {X 0,Y 530.601,Z 466.699,A -85,B 0,C 180,E1 -4402.388,E2 -4402.388} C_VEL
LIN {X 0,Y 530.529,Z 472.162,A -85,B 0,C 180,E1 -4403.916,E2 -4403.916} C_VEL
LIN {X 0,Y 530.413,Z 476.29,A -85,B 0,C 180,E1 -4405.44,E2 -4405.44} C_VEL
LIN {X 0,Y 530.448,Z 479.184,A -85,B 0,C 180,E1 -4406.962,E2 -4406.962} C_VEL
LIN {X 0,Y 530.358,Z 480.909,A -85,B 0,C 180,E1 -4408.481,E2 -4408.481} C_VEL
LIN {X 0,Y 530.34,Z 481.5,A -85,B 0,C 180,E1 -4410,E2 -4410} C_VEL
LIN {X 0,Y 530.358,Z 480.907,A -85,B 0,C 180,E1 -4411.518,E2 -4411.518} C_VEL
LIN {X 0,Y 530.448,Z 479.18,A -85,B 0,C 180,E1 -4413.038,E2 -4413.038} C_VEL
LIN {X 0,Y 530.412,Z 476.289,A -85,B 0,C 180,E1 -4414.559,E2 -4414.559} C_VEL
LIN {X 0,Y 530.533,Z 472.167,A -85,B 0,C 180,E1 -4416.083,E2 -4416.083} C_VEL
LIN {X 0,Y 530.6,Z 466.702,A -85,B 0,C 180,E1 -4417.611,E2 -4417.611} C_VEL
LIN {X 0,Y 530.759,Z 459.746,A -85,B 0,C 180,E1 -4419.142,E2 -4419.142} C_VEL
LIN {X 0,Y 531,Z 451.084,A -85,B 0,C 180,E1 -4420.678,E2 -4420.678} C_VEL
LIN {X 0,Y 531.229,Z 441.686,A -85,B 0,C 180,E1 -4422.051,E2 -4422.051} C_VEL
LIN {X 0,Y 531.563,Z 432.512,A -85,B 0,C 180,E1 -4423.183,E2 -4423.183} C_VEL
LIN {X 0,Y 531.961,Z 420.367,A -85,B 0,C 180,E1 -4424.44,E2 -4424.44} C_VEL
LIN {X 0,Y 532.386,Z 408.127,A -85,B 0,C 180,E1 -4425.492,E2 -4425.492} C_VEL
LIN {X 0,Y 532.766,Z 395.747,A -85,B 0,C 180,E1 -4426.377,E2 -4426.377} C_VEL
LIN {X 0,Y 533.191,Z 382.554,A -85,B 0,C 180,E1 -4427.152,E2 -4427.152} C_VEL
LIN {X 0,Y 533.612,Z 369.305,A -85,B 0,C 180,E1 -4427.779,E2 -4427.779} C_VEL
LIN {X 0,Y 533.927,Z 354.602,A -85,B 0,C 180,E1 -4428.32,E2 -4428.32} C_VEL
LIN {X 0,Y 534.012,Z 340.844,A -85,B 0,C 180,E1 -4428.691,E2 -4428.691} C_VEL
LIN {X 0,Y 530.596,Z 326.94,A -85,B 0,C 180,E1 -4429.086,E2 -4429.086} C_VEL
LIN {X 0,Y 530.669,Z 320.462,A -85,B 0,C 180,E1 -4432.02,E2 -4432.02} C_VEL
LIN {X 0,Y 530.722,Z 313.856,A -85,B 0,C 180,E1 -4435.071,E2 -4435.071} C_VEL
LIN {X 0,Y 530.817,Z 308.491,A -85,B 0,C 180,E1 -4437.606,E2 -4437.606} C_VEL
LIN {X 0,Y 530.921,Z 303.142,A -85,B 0,C 180,E1 -4440.199,E2 -4440.199} C_VEL
LIN {X 0,Y 531.091,Z 296.485,A -85,B 0,C 180,E1 -4443.521,E2 -4443.521} C_VEL
LIN {X 0,Y 531.189,Z 290.683,A -85,B 0,C 180,E1 -4446.539,E2 -4446.539} C_VEL
LIN {X 0,Y 531.313,Z 285.362,A -85,B 0,C 180,E1 -4449.413,E2 -4449.413} C_VEL
LIN {X 0,Y 531.333,Z 281.83,A -85,B 0,C 180,E1 -4451.402,E2 -4451.402} C_VEL
LIN {X 0,Y 531.01,Z 278.969,A -85,B 0,C 180,E1 -4453.148,E2 -4453.148} C_VEL
LIN {X 0,Y 530.978,Z 278.973,A -85,B 0,C 180,E1 -4455.621,E2 -4455.621} C_VEL
LIN {X 0,Y 530.989,Z 278.972,A -85,B 0,C 180,E1 -4458.564,E2 -4458.564} C_VEL
LIN {X 0,Y 530.954,Z 278.975,A -85,B 0,C 180,E1 -4461.529,E2 -4461.529} C_VEL
LIN {X 0,Y 530.941,Z 278.975,A -85,B 0,C 180,E1 -4464.379,E2 -4464.379} C_VEL
LIN {X 0,Y 530.964,Z 278.971,A -85,B 0,C 180,E1 -4467.133,E2 -4467.133} C_VEL
LIN {X 0,Y 530.961,Z 278.973,A -85,B 0,C 180,E1 -4469.803,E2 -4469.803} C_VEL
LIN {X 0,Y 531.001,Z 278.971,A -85,B 0,C 180,E1 -4472.468,E2 -4472.468} C_VEL
LIN {X 0,Y 530.998,Z 278.966,A -85,B 0,C 180,E1 -4474.942,E2 -4474.942} C_VEL
LIN {X 0,Y 530.962,Z 278.972,A -85,B 0,C 180,E1 -4478.246,E2 -4478.246} C_VEL
LIN {X 0,Y 530.988,Z 278.967,A -85,B 0,C 180,E1 -4480.677,E2 -4480.677} C_VEL
LIN {X 0,Y 530.977,Z 278.972,A -85,B 0,C 180,E1 -4483.071,E2 -4483.071} C_VEL
LIN {X 0,Y 531.006,Z 278.963,A -85,B 0,C 180,E1 -4485.436,E2 -4485.436} C_VEL
LIN {X 0,Y 531.039,Z 278.96,A -85,B 0,C 180,E1 -4488.55,E2 -4488.55} C_VEL
LIN {X 0,Y 531.045,Z 278.959,A -85,B 0,C 180,E1 -4491.629,E2 -4491.629} C_VEL
LIN {X 0,Y 531.112,Z 278.95,A -85,B 0,C 180,E1 -4494.685,E2 -4494.685} C_VEL
LIN {X 0,Y 531.135,Z 278.947,A -85,B 0,C 180,E1 -4497.725,E2 -4497.725} C_VEL
LIN {X 0,Y 531.138,Z 278.948,A -85,B 0,C 180,E1 -4500.758,E2 -4500.758} C_VEL
LIN {X 0,Y 531.1,Z 278.958,A -85,B 0,C 180,E1 -4503.034,E2 -4503.034} C_VEL
LIN {X 0,Y 531.059,Z 278.963,A -85,B 0,C 180,E1 -4506.077,E2 -4506.077} C_VEL
LIN {X 0,Y 531.023,Z 278.966,A -85,B 0,C 180,E1 -4509.138,E2 -4509.138} C_VEL
LIN {X 0,Y 531.031,Z 278.965,A -85,B 0,C 180,E1 -4512.225,E2 -4512.225} C_VEL
LIN {X 0,Y 530.985,Z 278.972,A -85,B 0,C 180,E1 -4515.35,E2 -4515.35} C_VEL
LIN {X 0,Y 530.985,Z 278.971,A -85,B 0,C 180,E1 -4518.521,E2 -4518.521} C_VEL
LIN {X 0,Y 530.99,Z 278.967,A -85,B 0,C 180,E1 -4520.938,E2 -4520.938} C_VEL
LIN {X 0,Y 530.973,Z 278.971,A -85,B 0,C 180,E1 -4524.225,E2 -4524.225} C_VEL
LIN {X 0,Y 530.992,Z 278.965,A -85,B 0,C 180,E1 -4526.744,E2 -4526.744} C_VEL
LIN {X 0,Y 530.973,Z 278.97,A -85,B 0,C 180,E1 -4529.323,E2 -4529.323} C_VEL
LIN {X 0,Y 530.973,Z 278.972,A -85,B 0,C 180,E1 -4532.103,E2 -4532.103} C_VEL
LIN {X 0,Y 530.959,Z 278.971,A -85,B 0,C 180,E1 -4534.851,E2 -4534.851} C_VEL
LIN {X 0,Y 530.959,Z 278.97,A -85,B 0,C 180,E1 -4537.508,E2 -4537.508} C_VEL
LIN {X 0,Y 530.978,Z 278.969,A -85,B 0,C 180,E1 -4540.433,E2 -4540.433} C_VEL
LIN {X 0,Y 530.956,Z 278.972,A -85,B 0,C 180,E1 -4543.282,E2 -4543.282} C_VEL
LIN {X 0,Y 530.948,Z 278.972,A -85,B 0,C 180,E1 -4543.548,E2 -4543.548} C_VEL
LIN {X 0,Y 530.279,Z 279.059,A -85,B 0,C 180,E1 -4544.181,E2 -4544.181} C_VEL
LIN {X 0,Y 527.439,Z 279.412,A -85,B 0,C 180,E1 -4545.21,E2 -4545.21} C_VEL
LIN {X 0,Y 525.033,Z 279.713,A -85,B 0,C 180,E1 -4546.039,E2 -4546.039} C_VEL
LIN {X 0,Y 523.989,Z 279.842,A -85,B 0,C 180,E1 -4546.678,E2 -4546.678} C_VEL
LIN {X 0,Y 523.898,Z 279.853,A -85,B 0,C 180,E1 -4546.895,E2 -4546.895} C_VEL
LIN {X 0,Y 523.898,Z 279.855,A -85,B 0,C 180,E1 -4547.546,E2 -4547.546} C_VEL
LIN {X 0,Y 524.058,Z 283.108,A -85,B 0,C 180,E1 -4549.855,E2 -4549.855} C_VEL
LIN {X 0,Y 523.992,Z 287.709,A -85,B 0,C 180,E1 -4552.876,E2 -4552.876} C_VEL
LIN {X 0,Y 523.914,Z 292.164,A -85,B 0,C 180,E1 -4555.709,E2 -4555.709} C_VEL
LIN {X 0,Y 523.783,Z 296.609,A -85,B 0,C 180,E1 -4558.448,E2 -4558.448} C_VEL
LIN {X 0,Y 523.732,Z 301.047,A -85,B 0,C 180,E1 -4561.114,E2 -4561.114} C_VEL
LIN {X 0,Y 523.644,Z 306.085,A -85,B 0,C 180,E1 -4564.057,E2 -4564.057} C_VEL
LIN {X 0,Y 523.591,Z 309.951,A -85,B 0,C 180,E1 -4566.255,E2 -4566.255} C_VEL
LIN {X 0,Y 523.48,Z 315.853,A -85,B 0,C 180,E1 -4569.571,E2 -4569.571} C_VEL
LIN {X 0,Y 523.489,Z 317.953,A -85,B 0,C 180,E1 -4570.717,E2 -4570.717} C_VEL
LIN {X 0,Y 527.418,Z 333.647,A -85,B 0,C 180,E1 -4571.168,E2 -4571.168} C_VEL
LIN {X 0,Y 527.148,Z 348.746,A -85,B 0,C 180,E1 -4571.611,E2 -4571.611} C_VEL
LIN {X 0,Y 526.699,Z 364.052,A -85,B 0,C 180,E1 -4572.228,E2 -4572.228} C_VEL
LIN {X 0,Y 526.224,Z 378.912,A -85,B 0,C 180,E1 -4573.014,E2 -4573.014} C_VEL
LIN {X 0,Y 525.748,Z 392.321,A -85,B 0,C 180,E1 -4573.897,E2 -4573.897} C_VEL
LIN {X 0,Y 525.242,Z 404.594,A -85,B 0,C 180,E1 -4574.876,E2 -4574.876} C_VEL
LIN {X 0,Y 524.778,Z 416.83,A -85,B 0,C 180,E1 -4576.051,E2 -4576.051} C_VEL
LIN {X 0,Y 524.391,Z 427.057,A -85,B 0,C 180,E1 -4577.225,E2 -4577.225} C_VEL
LIN {X 0,Y 524.052,Z 437.07,A -85,B 0,C 180,E1 -4578.592,E2 -4578.592} C_VEL
LIN {X 0,Y 523.782,Z 445.387,A -85,B 0,C 180,E1 -4579.955,E2 -4579.955} C_VEL
LIN {X 0,Y 523.614,Z 453.212,A -85,B 0,C 180,E1 -4581.51,E2 -4581.51} C_VEL
LIN {X 0,Y 523.482,Z 459.445,A -85,B 0,C 180,E1 -4583.06,E2 -4583.06} C_VEL
LIN {X 0,Y 523.441,Z 464.263,A -85,B 0,C 180,E1 -4584.607,E2 -4584.607} C_VEL
LIN {X 0,Y 523.402,Z 467.798,A -85,B 0,C 180,E1 -4586.151,E2 -4586.151} C_VEL
LIN {X 0,Y 523.333,Z 470.139,A -85,B 0,C 180,E1 -4587.691,E2 -4587.691} C_VEL
LIN {X 0,Y 523.246,Z 471.337,A -85,B 0,C 180,E1 -4589.231,E2 -4589.231} C_VEL
LIN {X 0,Y 523.247,Z 471.357,A -85,B 0,C 180,E1 -4590.77,E2 -4590.77} C_VEL
LIN {X 0,Y 523.333,Z 470.235,A -85,B 0,C 180,E1 -4592.309,E2 -4592.309} C_VEL
LIN {X 0,Y 523.402,Z 467.971,A -85,B 0,C 180,E1 -4593.85,E2 -4593.85} C_VEL
LIN {X 0,Y 523.438,Z 464.509,A -85,B 0,C 180,E1 -4595.393,E2 -4595.393} C_VEL
LIN {X 0,Y 523.482,Z 459.77,A -85,B 0,C 180,E1 -4596.94,E2 -4596.94} C_VEL
LIN {X 0,Y 523.613,Z 453.631,A -85,B 0,C 180,E1 -4598.491,E2 -4598.491} C_VEL
LIN {X 0,Y 523.776,Z 445.904,A -85,B 0,C 180,E1 -4600.046,E2 -4600.046} C_VEL
LIN {X 0,Y 524.003,Z 437.676,A -85,B 0,C 180,E1 -4601.41,E2 -4601.41} C_VEL
LIN {X 0,Y 524.355,Z 427.782,A -85,B 0,C 180,E1 -4602.777,E2 -4602.777} C_VEL
LIN {X 0,Y 524.745,Z 417.639,A -85,B 0,C 180,E1 -4603.95,E2 -4603.95} C_VEL
LIN {X 0,Y 525.203,Z 405.704,A -85,B 0,C 180,E1 -4605.113,E2 -4605.113} C_VEL
LIN {X 0,Y 525.714,Z 392.309,A -85,B 0,C 180,E1 -4606.195,E2 -4606.195} C_VEL
LIN {X 0,Y 526.225,Z 378.751,A -85,B 0,C 180,E1 -4607.087,E2 -4607.087} C_VEL
LIN {X 0,Y 526.659,Z 364.845,A -85,B 0,C 180,E1 -4607.824,E2 -4607.824} C_VEL
LIN {X 0,Y 527.085,Z 349.552,A -85,B 0,C 180,E1 -4608.452,E2 -4608.452} C_VEL
LIN {X 0,Y 527.457,Z 333.727,A -85,B 0,C 180,E1 -4608.918,E2 -4608.918} C_VEL
LIN {X 0,Y 523.495,Z 317.917,A -85,B 0,C 180,E1 -4609.38,E2 -4609.38} C_VEL
LIN {X 0,Y 523.532,Z 311.602,A -85,B 0,C 180,E1 -4612.911,E2 -4612.911} C_VEL
LIN {X 0,Y 523.645,Z 306.3,A -85,B 0,C 180,E1 -4615.943,E2 -4615.943} C_VEL
LIN {X 0,Y 523.732,Z 301.238,A -85,B 0,C 180,E1 -4618.887,E2 -4618.887} C_VEL
LIN {X 0,Y 523.805,Z 296.779,A -85,B 0,C 180,E1 -4621.552,E2 -4621.552} C_VEL
LIN {X 0,Y 523.916,Z 292.309,A -85,B 0,C 180,E1 -4624.291,E2 -4624.291} C_VEL
LIN {X 0,Y 523.995,Z 287.841,A -85,B 0,C 180,E1 -4627.125,E2 -4627.125} C_VEL
LIN {X 0,Y 524.061,Z 283.25,A -85,B 0,C 180,E1 -4630.146,E2 -4630.146} C_VEL
LIN {X 0,Y 523.901,Z 279.895,A -85,B 0,C 180,E1 -4632.455,E2 -4632.455} C_VEL
LIN {X 0,Y 523.953,Z 279.847,A -85,B 0,C 180,E1 -4635.309,E2 -4635.309} C_VEL
LIN {X 0,Y 523.954,Z 279.847,A -85,B 0,C 180,E1 -4638.69,E2 -4638.69} C_VEL
LIN {X 0,Y 523.919,Z 279.848,A -85,B 0,C 180,E1 -4641.08,E2 -4641.08} C_VEL
LIN {X 0,Y 523.894,Z 279.852,A -85,B 0,C 180,E1 -4643.825,E2 -4643.825} C_VEL
LIN {X 0,Y 523.938,Z 279.848,A -85,B 0,C 180,E1 -4646.635,E2 -4646.635} C_VEL
LIN {X 0,Y 523.954,Z 279.848,A -85,B 0,C 180,E1 -4649.355,E2 -4649.355} C_VEL
LIN {X 0,Y 523.941,Z 279.847,A -85,B 0,C 180,E1 -4652.288,E2 -4652.288} C_VEL
LIN {X 0,Y 523.924,Z 279.85,A -85,B 0,C 180,E1 -4655.428,E2 -4655.428} C_VEL
LIN {X 0,Y 523.935,Z 279.844,A -85,B 0,C 180,E1 -4657.939,E2 -4657.939} C_VEL
LIN {X 0,Y 523.971,Z 279.843,A -85,B 0,C 180,E1 -4660.408,E2 -4660.408} C_VEL
LIN {X 0,Y 523.963,Z 279.843,A -85,B 0,C 180,E1 -4662.837,E2 -4662.837} C_VEL
LIN {X 0,Y 523.969,Z 279.842,A -85,B 0,C 180,E1 -4665.235,E2 -4665.235} C_VEL
LIN {X 0,Y 524.009,Z 279.836,A -85,B 0,C 180,E1 -4668.394,E2 -4668.394} C_VEL
LIN {X 0,Y 523.999,Z 279.837,A -85,B 0,C 180,E1 -4671.516,E2 -4671.516} C_VEL
LIN {X 0,Y 524.074,Z 279.828,A -85,B 0,C 180,E1 -4674.613,E2 -4674.613} C_VEL
LIN {X 0,Y 524.11,Z 279.823,A -85,B 0,C 180,E1 -4677.694,E2 -4677.694} C_VEL
LIN {X 0,Y 524.112,Z 279.823,A -85,B 0,C 180,E1 -4680.768,E2 -4680.768} C_VEL
LIN {X 0,Y 524.07,Z 279.833,A -85,B 0,C 180,E1 -4683.075,E2 -4683.075} C_VEL
LIN {X 0,Y 524.02,Z 279.84,A -85,B 0,C 180,E1 -4686.159,E2 -4686.159} C_VEL
LIN {X 0,Y 523.994,Z 279.843,A -85,B 0,C 180,E1 -4689.262,E2 -4689.262} C_VEL
LIN {X 0,Y 523.999,Z 279.838,A -85,B 0,C 180,E1 -4691.739,E2 -4691.739} C_VEL
LIN {X 0,Y 523.987,Z 279.841,A -85,B 0,C 180,E1 -4695.052,E2 -4695.052} C_VEL
LIN {X 0,Y 523.96,Z 279.843,A -85,B 0,C 180,E1 -4697.969,E2 -4697.969} C_VEL
LIN {X 0,Y 523.953,Z 279.844,A -85,B 0,C 180,E1 -4700.411,E2 -4700.411} C_VEL
LIN {X 0,Y 523.907,Z 279.853,A -85,B 0,C 180,E1 -4702.894,E2 -4702.894} C_VEL
LIN {X 0,Y 523.949,Z 279.843,A -85,B 0,C 180,E1 -4705.419,E2 -4705.419} C_VEL
LIN {X 0,Y 523.952,Z 279.845,A -85,B 0,C 180,E1 -4708,E2 -4708} C_VEL
LIN {X 0,Y 523.936,Z 279.85,A -85,B 0,C 180,E1 -4710.854,E2 -4710.854} C_VEL
LIN {X 0,Y 523.955,Z 279.85,A -85,B 0,C 180,E1 -4713.734,E2 -4713.734} C_VEL
LIN {X 0,Y 523.896,Z 279.854,A -85,B 0,C 180,E1 -4716.401,E2 -4716.401} C_VEL
LIN {X 0,Y 523.921,Z 279.849,A -85,B 0,C 180,E1 -4719.085,E2 -4719.085} C_VEL
LIN {X 0,Y 523.939,Z 279.846,A -85,B 0,C 180,E1 -4722.12,E2 -4722.12} C_VEL
LIN {X 0,Y 523.954,Z 279.849,A -85,B 0,C 180,E1 -4725.309,E2 -4725.309} C_VEL
LIN {X 0,Y 524.002,Z 280.051,A -85,B 0,C 180,E1 -4726.842,E2 -4726.842} C_VEL
LIN {X 0,Y 524.359,Z 283.575,A -85,B 0,C 180,E1 -4728.948,E2 -4728.948} C_VEL
LIN {X 0,Y 524.238,Z 288.873,A -85,B 0,C 180,E1 -4731.926,E2 -4731.926} C_VEL
LIN {X 0,Y 524.121,Z 294.371,A -85,B 0,C 180,E1 -4734.881,E2 -4734.881} C_VEL
LIN {X 0,Y 523.957,Z 299.763,A -85,B 0,C 180,E1 -4737.676,E2 -4737.676} C_VEL
LIN {X 0,Y 523.849,Z 305.776,A -85,B 0,C 180,E1 -4740.697,E2 -4740.697} C_VEL
LIN {X 0,Y 523.696,Z 311.993,A -85,B 0,C 180,E1 -4743.714,E2 -4743.714} C_VEL
LIN {X 0,Y 523.638,Z 317.365,A -85,B 0,C 180,E1 -4746.256,E2 -4746.256} C_VEL
LIN {X 0,Y 523.562,Z 322.726,A -85,B 0,C 180,E1 -4748.75,E2 -4748.75} C_VEL
LIN {X 0,Y 523.575,Z 327.025,A -85,B 0,C 180,E1 -4750.668,E2 -4750.668} C_VEL
LIN {X 0,Y 527.409,Z 342.506,A -85,B 0,C 180,E1 -4751.104,E2 -4751.104} C_VEL
LIN {X 0,Y 527.125,Z 357.868,A -85,B 0,C 180,E1 -4751.546,E2 -4751.546} C_VEL
LIN {X 0,Y 526.666,Z 372.557,A -85,B 0,C 180,E1 -4752.126,E2 -4752.126} C_VEL
LIN {X 0,Y 526.249,Z 386.017,A -85,B 0,C 180,E1 -4752.814,E2 -4752.814} C_VEL
LIN {X 0,Y 525.774,Z 399.951,A -85,B 0,C 180,E1 -4753.698,E2 -4753.698} C_VEL
LIN {X 0,Y 525.305,Z 412.62,A -85,B 0,C 180,E1 -4754.679,E2 -4754.679} C_VEL
LIN {X 0,Y 524.897,Z 423.273,A -85,B 0,C 180,E1 -4755.658,E2 -4755.658} C_VEL
LIN {X 0,Y 524.508,Z 434.107,A -85,B 0,C 180,E1 -4756.833,E2 -4756.833} C_VEL
LIN {X 0,Y 524.137,Z 443.298,A -85,B 0,C 180,E1 -4758.005,E2 -4758.005} C_VEL
LIN {X 0,Y 523.943,Z 452.296,A -85,B 0,C 180,E1 -4759.372,E2 -4759.372} C_VEL
LIN {X 0,Y 523.699,Z 459.748,A -85,B 0,C 180,E1 -4760.733,E2 -4760.733} C_VEL
LIN {X 0,Y 523.535,Z 466.699,A -85,B 0,C 180,E1 -4762.285,E2 -4762.285} C_VEL
LIN {X 0,Y 523.441,Z 472.161,A -85,B 0,C 180,E1 -4763.834,E2 -4763.834} C_VEL
LIN {X 0,Y 523.323,Z 476.29,A -85,B 0,C 180,E1 -4765.378,E2 -4765.378} C_VEL
LIN {X 0,Y 523.358,Z 479.183,A -85,B 0,C 180,E1 -4766.921,E2 -4766.921} C_VEL
LIN {X 0,Y 523.272,Z 480.909,A -85,B 0,C 180,E1 -4768.46,E2 -4768.46} C_VEL
LIN {X 0,Y 523.243,Z 481.5,A -85,B 0,C 180,E1 -4770,E2 -4770} C_VEL
LIN {X 0,Y 523.272,Z 480.907,A -85,B 0,C 180,E1 -4771.539,E2 -4771.539} C_VEL
LIN {X 0,Y 523.358,Z 479.179,A -85,B 0,C 180,E1 -4773.079,E2 -4773.079} C_VEL
LIN {X 0,Y 523.323,Z 476.289,A -85,B 0,C 180,E1 -4774.621,E2 -4774.621} C_VEL
LIN {X 0,Y 523.45,Z 472.167,A -85,B 0,C 180,E1 -4776.166,E2 -4776.166} C_VEL
LIN {X 0,Y 523.534,Z 466.702,A -85,B 0,C 180,E1 -4777.714,E2 -4777.714} C_VEL
LIN {X 0,Y 523.698,Z 459.745,A -85,B 0,C 180,E1 -4779.267,E2 -4779.267} C_VEL
LIN {X 0,Y 523.986,Z 451.083,A -85,B 0,C 180,E1 -4780.823,E2 -4780.823} C_VEL
LIN {X 0,Y 524.231,Z 441.836,A -85,B 0,C 180,E1 -4782.193,E2 -4782.193} C_VEL
LIN {X 0,Y 524.598,Z 432.479,A -85,B 0,C 180,E1 -4783.361,E2 -4783.361} C_VEL
LIN {X 0,Y 525.037,Z 420.31,A -85,B 0,C 180,E1 -4784.634,E2 -4784.634} C_VEL
LIN {X 0,Y 525.481,Z 408.755,A -85,B 0,C 180,E1 -4785.644,E2 -4785.644} C_VEL
LIN {X 0,Y 525.9,Z 395.677,A -85,B 0,C 180,E1 -4786.597,E2 -4786.597} C_VEL
LIN {X 0,Y 526.38,Z 382.484,A -85,B 0,C 180,E1 -4787.381,E2 -4787.381} C_VEL
LIN {X 0,Y 526.826,Z 369.38,A -85,B 0,C 180,E1 -4788.009,E2 -4788.009} C_VEL
LIN {X 0,Y 527.19,Z 354.533,A -85,B 0,C 180,E1 -4788.562,E2 -4788.562} C_VEL
LIN {X 0,Y 527.264,Z 341.97,A -85,B 0,C 180,E1 -4788.913,E2 -4788.913} C_VEL
LIN {X 0,Y 523.545,Z 326.881,A -85,B 0,C 180,E1 -4789.347,E2 -4789.347} C_VEL
LIN {X 0,Y 523.604,Z 320.792,A -85,B 0,C 180,E1 -4792.159,E2 -4792.159} C_VEL
LIN {X 0,Y 523.654,Z 315.602,A -85,B 0,C 180,E1 -4794.585,E2 -4794.585} C_VEL
LIN {X 0,Y 523.769,Z 309.141,A -85,B 0,C 180,E1 -4797.675,E2 -4797.675} C_VEL
LIN {X 0,Y 523.908,Z 303.099,A -85,B 0,C 180,E1 -4800.647,E2 -4800.647} C_VEL
LIN {X 0,Y 524.051,Z 296.99,A -85,B 0,C 180,E1 -4803.749,E2 -4803.749} C_VEL
LIN {X 0,Y 524.169,Z 291.884,A -85,B 0,C 180,E1 -4806.441,E2 -4806.441} C_VEL
LIN {X 0,Y 524.289,Z 287.106,A -85,B 0,C 180,E1 -4809.051,E2 -4809.051} C_VEL
LIN {X 0,Y 524.338,Z 283.036,A -85,B 0,C 180,E1 -4811.358,E2 -4811.358} C_VEL
LIN {X 0,Y 523.97,Z 279.845,A -85,B 0,C 180,E1 -4813.372,E2 -4813.372} C_VEL
LIN {X 0,Y 523.913,Z 279.85,A -85,B 0,C 180,E1 -4816.416,E2 -4816.416} C_VEL
LIN {X 0,Y 523.935,Z 279.849,A -85,B 0,C 180,E1 -4818.907,E2 -4818.907} C_VEL
LIN {X 0,Y 523.911,Z 279.853,A -85,B 0,C 180,E1 -4821.898,E2 -4821.898} C_VEL
LIN {X 0,Y 523.914,Z 279.854,A -85,B 0,C 180,E1 -4824.911,E2 -4824.911} C_VEL
LIN {X 0,Y 523.935,Z 279.85,A -85,B 0,C 180,E1 -4827.678,E2 -4827.678} C_VEL
LIN {X 0,Y 523.945,Z 279.848,A -85,B 0,C 180,E1 -4830.676,E2 -4830.676} C_VEL
LIN {X 0,Y 523.965,Z 279.845,A -85,B 0,C 180,E1 -4833.728,E2 -4833.728} C_VEL
LIN {X 0,Y 523.928,Z 279.846,A -85,B 0,C 180,E1 -4836.27,E2 -4836.27} C_VEL
LIN {X 0,Y 523.937,Z 279.848,A -85,B 0,C 180,E1 -4838.766,E2 -4838.766} C_VEL
LIN {X 0,Y 523.945,Z 279.845,A -85,B 0,C 180,E1 -4841.221,E2 -4841.221} C_VEL
LIN {X 0,Y 523.927,Z 279.847,A -85,B 0,C 180,E1 -4843.639,E2 -4843.639} C_VEL
LIN {X 0,Y 523.925,Z 279.849,A -85,B 0,C 180,E1 -4846.028,E2 -4846.028} C_VEL
LIN {X 0,Y 524.003,Z 279.836,A -85,B 0,C 180,E1 -4848.394,E2 -4848.394} C_VEL
LIN {X 0,Y 523.994,Z 279.837,A -85,B 0,C 180,E1 -4851.516,E2 -4851.516} C_VEL
LIN {X 0,Y 524.072,Z 279.827,A -85,B 0,C 180,E1 -4854.614,E2 -4854.614} C_VEL
LIN {X 0,Y 524.107,Z 279.822,A -85,B 0,C 180,E1 -4857.695,E2 -4857.695} C_VEL
LIN {X 0,Y 524.109,Z 279.823,A -85,B 0,C 180,E1 -4860.768,E2 -4860.768} C_VEL
LIN {X 0,Y 524.067,Z 279.834,A -85,B 0,C 180,E1 -4863.075,E2 -4863.075} C_VEL
LIN {X 0,Y 524.017,Z 279.84,A -85,B 0,C 180,E1 -4866.159,E2 -4866.159} C_VEL
LIN {X 0,Y 523.991,Z 279.843,A -85,B 0,C 180,E1 -4869.262,E2 -4869.262} C_VEL
LIN {X 0,Y 523.994,Z 279.837,A -85,B 0,C 180,E1 -4871.74,E2 -4871.74} C_VEL
LIN {X 0,Y 523.983,Z 279.841,A -85,B 0,C 180,E1 -4875.052,E2 -4875.052} C_VEL
LIN {X 0,Y 523.956,Z 279.843,A -85,B 0,C 180,E1 -4877.969,E2 -4877.969} C_VEL
LIN {X 0,Y 523.963,Z 279.842,A -85,B 0,C 180,E1 -4880.41,E2 -4880.41} C_VEL
LIN {X 0,Y 523.909,Z 279.853,A -85,B 0,C 180,E1 -4882.894,E2 -4882.894} C_VEL
LIN {X 0,Y 523.945,Z 279.844,A -85,B 0,C 180,E1 -4885.419,E2 -4885.419} C_VEL
LIN {X 0,Y 523.949,Z 279.843,A -85,B 0,C 180,E1 -4888,E2 -4888} C_VEL
LIN {X 0,Y 523.94,Z 279.846,A -85,B 0,C 180,E1 -4890.856,E2 -4890.856} C_VEL
LIN {X 0,Y 523.951,Z 279.847,A -85,B 0,C 180,E1 -4893.735,E2 -4893.735} C_VEL
LIN {X 0,Y 523.893,Z 279.852,A -85,B 0,C 180,E1 -4896.401,E2 -4896.401} C_VEL
LIN {X 0,Y 523.918,Z 279.848,A -85,B 0,C 180,E1 -4899.085,E2 -4899.085} C_VEL
LIN {X 0,Y 523.947,Z 279.845,A -85,B 0,C 180,E1 -4902.12,E2 -4902.12} C_VEL
LIN {X 0,Y 523.951,Z 279.844,A -85,B 0,C 180,E1 -4905.309,E2 -4905.309} C_VEL
LIN {X 0,Y 523.898,Z 279.853,A -85,B 0,C 180,E1 -4906.895,E2 -4906.895} C_VEL
LIN {X 0,Y 523.226,Z 280.198,A -85,B 0,C 180,E1 -4907.535,E2 -4907.535} C_VEL
LIN {X 0,Y 520.429,Z 281.748,A -85,B 0,C 180,E1 -4908.566,E2 -4908.566} C_VEL
